// TIA Portal V20 program export: 1 tag tables, 0 data types, 3 data blocks, 33 code blocks (in call order from the OBs), 11 instance data blocks

VAR_GLOBAL   // PLC tag table "Default tag table"
   Doser1 AT %I0.0 : Bool;
   AlarmOpen1 AT %I0.1 : Bool;
   Doser2 AT %I0.2 : Bool;
   AlarmOpen2 AT %I0.3 : Bool;
   RunClose1 AT %I0.4 : Bool;
   RunOpen1 AT %I0.5 : Bool;
   RunClose2 AT %I0.6 : Bool;
   RunOpen2 AT %I0.7 : Bool;
   WaterCounterInPulse AT %I1.0 : Bool;
   WaterCounterOutPulse AT %I1.1 : Bool;
   AI0V AT %IW64 : Int;
   AI1V AT %IW66 : Int;
   AI0AV AT %IW128 : Int;
   AI1AV AT %IW130 : Int;
   AI2AV AT %IW132 : Int;
   AI3AV AT %IW134 : Int;
   AI4AV AT %IW80 : Int;
   PowerSupply AT %I1.2 : Bool;
   FlowAO AT %QW64 : Int;
   OutOpen1 AT %Q0.0 : Bool;
   OutClose1 AT %Q0.1 : Bool;
   OutOpen2 AT %Q0.2 : Bool;
   OutClose2 AT %Q0.3 : Bool;
   SirenOut AT %Q0.4 : Bool;
   System_Byte AT %MB1 : Byte;
   FirstScan AT %M1.0 : Bool;
   DiagStatusUpdate AT %M1.1 : Bool;
   AlwaysTRUE AT %M1.2 : Bool;
   AlwaysFALSE AT %M1.3 : Bool;
   Clock_Byte AT %MB0 : Byte;
   Clock_10Hz AT %M0.0 : Bool;
   Clock_5Hz AT %M0.1 : Bool;
   "Clock_2.5Hz" AT %M0.2 : Bool;
   Clock_2Hz AT %M0.3 : Bool;
   "Clock_1.25Hz" AT %M0.4 : Bool;
   Clock_1Hz AT %M0.5 : Bool;
   "Clock_0.625Hz" AT %M0.6 : Bool;
   "Clock_0.5Hz" AT %M0.7 : Bool;
   Damper1_AutoMode AT %I1.3 : Bool;
   Damper2_AutoMode AT %I1.4 : Bool;
   OsmosOut AT %Q0.5 : Bool;
   OsmosAO AT %QW66 : Int;
   DoserOut AT %Q0.6 : Bool;
   ChlorationOut AT %Q0.7 : Bool;
END_VAR

DATA_BLOCK "Config"   // DB20
{ S7_Optimized_Access := 'FALSE' }
VERSION : 0.1
// stored: AutoNumber false, DBAccessibleFromOPCUA true, IsOnlyStoredInLoadMemory false, IsWriteProtectedInAS false
   VAR
      DateTime : DTL := DTL#2024-10-30-11:20:02.078798;
      HMI_ResetWaterCounter : Bool := FALSE;
      HMI_ResetPositionDamper1 : Bool := FALSE;
      HMI_ResetPositionDamper2 : Bool := FALSE;
      HMI_StartAdjustDamper1 : Bool := FALSE;
      HMI_StartAdjustDamper2 : Bool := FALSE;
      HMI_StopAdjustDamper1 : Bool := FALSE;
      HMI_StopAdjustDamper2 : Bool := FALSE;
      HMI_WeightToZero : Bool := FALSE;
      WaterPulseDuble : Bool;
      DiOxydeDosing : DWord;
   END_VAR
BEGIN
END_DATA_BLOCK

DATA_BLOCK "MB"   // DB1
{ S7_Optimized_Access := 'FALSE' }
VERSION : 0.1
// stored: AutoNumber false, DBAccessibleFromOPCUA true, IsOnlyStoredInLoadMemory false, IsWriteProtectedInAS false
   VAR RETAIN
      Table : Struct
         Service : Bool := FALSE;
         CycleDay : Int := 0;
         CycleStatus : Word := 16#0001;
         RestTimeC1 : UInt := 10;
         RestTimeC2 : UInt := 20;
         RestTimeC3 : UInt := 27;
         RestTimeC4 : UInt := 45;
         RestTimeC5 : UInt := 9999;
         CycleStartDay : Array[0..4] of UInt;
         LevelRCV1Min : Real := 190.0;
         LevelRCV1Max : Real := 210.0;
         LevelRCV2Min : Real := 190.0;
         LevelRCV2Max : Real := 210.0;
         LevelRCV1BasicMin : Real := 200.0;
         LevelRCV1BasicMax : Real := 250.0;
         LevelRCV2BasicMin : Real := 200.0;
         LevelRCV2BasicMax : Real := 250.0;
         LevelRCVCycle : Array[0..4] of Struct
            Min : Real;
            Max : Real;
         END_STRUCT;
         WaterCounterInPulseValue : Real := 0.1;
         WaterCounterInDailyValue : Real := 0.0;
         WaterCounterInTotalValue : Real := 0.0;
         AIOffsetCH0 : Real := 0.0;
         AIValueMinCH0 : Real := 0.0;
         AIValueMaxCH0 : Real := 1.0;
         AITimeBaseCH0 : Time := T#0MS;
         AIOffsetCH1 : Real := 0.0;
         AIValueMinCH1 : Real := 0.0;
         AIValueMaxCH1 : Real := 1200.0;
         AITimeBaseCH1 : Time := T#5MS;
         AIOffsetCH2 : Real := 0.0;
         AIValueMinCH2 : Real := 0.0;
         AIValueMaxCH2 : Real := 1200.0;
         AITimeBaseCH2 : Time := T#5MS;
         AIOffsetCH3 : Real := 0.0;
         AIValueMinCH3 : Real := 0.0;
         AIValueMaxCH3 : Real := 16.0;
         AITimeBaseCH3 : Time := T#2MS;
         AIOffsetCH4 : Real := 0.0;
         AIValueMinCH4 : Real := 0.0;
         AIValueMaxCH4 : Real := 16.0;
         AITimeBaseCH4 : Time := T#2MS;
         AIOffsetCH5 : Real := 0.0;
         AIValueMinCH5 : Real := 0.0;
         AIValueMaxCH5 : Real := 0.0;
         AITimeBaseCH5 : Time := T#0MS;
         ChlorValue : Real := 0.8276128;
         RCV1LevelValue : Real := 0.07552084;
         RCV2LevelValue : Real := 199.1832;
         WaterInPressureValue : Real := 0.0;
         WaterOutPressureValue : Real := 4.414607;
         Reserved : Real := 0.0;
         LevelRCV1AlarmMin : Real := 100.0;
         LevelRCV1AlarmMax : Real := 400.0;
         LevelRCV2AlarmMin : Real := 100.0;
         LevelRCV2AlarmMax : Real := 400.0;
         Chlor_Setpoint : Real := 0.0;
         Chlor_PulseWeight : Real := 0.0;
         Chlor_ConcentAlarm : Real := 0.9;
         Chlor_BaseDose : Real := 25.0;   // Була задача в ручному
         Chlor_SetpointMin : Real := 1.0;
         Chlor_SetpointMax : Real := 1.1;
         Chlor_Corection : Real := 0.5;
         Doser1_PulseValue : Real := 10.0;
         Reserved_2 : Int := 0;
         Reserved_3 : Int := 0;
         Doser1_DailyValue : Real := 0.0;
         Doser1_TotalValue : Real := 0.0;
         Doser1_Cunsumption : Real := 0.0;
         Doser2_PulseValue : Real := 0.81;
         Reserved_4 : Int := 0;
         Reserved_5 : Int := 0;
         Doser2_DailyValue : Real := 0.0;
         Doser2_TotalValue : Real := 0.0;
         Doser2_Cunsumption : Real := 0.0;
         PumpDoserValue : Real := 0.0;
         CalibratedPumpDoserValueMA : Real := 4.0;
         PumpDoserCalibrationMA : Real := 0.0;
         PumpDoserProductivity : Real := 6300.0;
         DampersSyncMode : Word := 16#0000;
         UsePID : Bool := FALSE;
         Damper1_PID_SetpointDeadZone : Real := 5.0;
         Damper1_PID_KP : Real := 2.0;
         Damper1_PID_KI : Real := 0.3;
         Damper1_PID_KD : Real := 0.1;
         Damper1_PID_TI : Real := 600.0;
         Damper1_PositionDeadZone : Real := 1.0;
         Damper1_FullMovingTime : Real := 26.14;
         Damper1_Position : Real := 0.0;
         Damper1_PositionSetpoint : Real := 100.0;
         Damper1_PID_Setpoint : Real := 200.0;
         Damper2_PID_SetpointDeadZone : Real := 5.0;
         Damper2_PID_KP : Real := 2.0;
         Damper2_PID_KI : Real := 0.3;
         Damper2_PID_KD : Real := 0.1;
         Damper2_PID_TI : Real := 600.0;
         Damper2_PositionDeadZone : Real := 1.0;
         Damper2_FullMovingTime : Real := 28.0;
         Damper2_Position : Real := 0.0;
         Damper2_PositionSetpoint : Real := 0.0;
         Damper2_PID_Setpoint : Real := 200.0;
         HMI_CycleOn : Bool := TRUE;
         HMI_ChlorModeOn : Bool := FALSE;
         HMI_Chlor_ChooseTank : Bool := TRUE;   // 0 - РЧВ1 1 -РЧВ2
         HMI_ManualModeOn : Bool := FALSE;
         HMI_SoundOff : Bool := TRUE;
         HMI_ManualOpenDamper1 : Bool := FALSE;
         HMI_ManualOpenDamper2 : Bool := FALSE;
         HMI_ResetWaterCounter : Bool := FALSE;
         HMI_ResetPositionDamper1 : Bool := FALSE;
         HMI_ResetPositionDamper2 : Bool := FALSE;
         HMI_StartAdjustDamper1 : Bool := FALSE;
         HMI_StartAdjustDamper2 : Bool := FALSE;
         HMI_StopAdjustDamper1 : Bool := FALSE;
         HMI_StopAdjustDamper2 : Bool := FALSE;
         HMI_WeightToZero : Bool := FALSE;
         HMI_WeightAlarmReset : Bool := FALSE;
         Alarms_Open1 : Bool := FALSE;
         Alarms_Open2 : Bool := FALSE;
         Alarms_ChlorLargeConsumption : Bool := FALSE;
         Alarms_RCV1Max : Bool := FALSE;
         Alarms_RCV1Min : Bool := TRUE;
         Alarms_RCV2Max : Bool := FALSE;
         Alarms_RCV2Min : Bool := FALSE;
         Alarms_RCV1Error : Bool := FALSE;
         Alarms_RCV2Error : Bool := FALSE;
         Alarms_ChlorMax : Bool := FALSE;
         Alarms_NoFlow : Bool := FALSE;
         Alarms_WaterOutMax : Bool := FALSE;
         Alarms_WaterOutMin : Bool := FALSE;
         Alarms_NoPowerSupply : Bool := FALSE;
         Alarms_WaterInMax : Bool := FALSE;
         Alarms_WaterInMin : Bool := FALSE;
         WaterOutMaxValue : Real := 6.0;
         WaterOutMinValue : Real := 1.5;
         WaterOutAlarmTime : DInt := 10;
         GlobalAlarm : Bool := FALSE;
         SensorWeightVoltage1 : Real := 1.681112;
         WeightValueMin1 : Real := 356.0;
         WeightValueMax1 : Real := 361.0;
         WeightValueOffset1 : Real := 0.0;
         WeightValue1 : Real := 353.3342;
         WeightVoltageMin1 : Real := 1.691255;
         WeightVoltageMax1 : Real := 1.71028;
         DayChangeFlag : Bool := TRUE;
         Damper1_AdjustBusy : Bool := FALSE;
         Damper1_AdjustError : Bool := FALSE;
         Damper1_AdjustDone : Bool := FALSE;
         Damper2_AdjustBusy : Bool := FALSE;
         Damper2_AdjustError : Bool := FALSE;
         Damper2_AdjustDone : Bool := FALSE;
         "Damper1_Close/Open" : Bool := FALSE;
         "Damper2_Close/Open" : Bool := FALSE;
         "Damper1_Manual/Auto" : Bool := FALSE;
         "Damper2_Manual/Auto" : Bool := TRUE;
         SensorWeightVoltage2 : Real := -0.2375481;
         WeightValueMin2 : Real := 0.0;
         WeightValueMax2 : Real := 5.0;
         WeightValueOffset2 : Real := 0.0;
         WeightValue2 : Real := 0.0;
         WeightVoltageMin2 : Real := 0.155;
         WeightVoltageMax2 : Real := 0.177;
         WaterConsumption : Real := 0.0;
         LevelRCV1AlarmMinBasic : Real := 0.0;
         LevelRCV1AlarmMaxBasic : Real := 0.0;
         LevelRCV2AlarmMinBasic : Real := 0.0;
         LevelRCV2AlarmMaxBasic : Real := 0.0;
         LevelRCV1AlarmDeltaC1 : Real := 20.0;
         LevelRCV1AlarmDeltaC2 : Real := 20.0;
         LevelRCV1AlarmDeltaC3 : Real := 20.0;
         LevelRCV1AlarmDeltaC4 : Real := 20.0;
         LevelRCV1AlarmDeltaC5 : Real := 20.0;
         LevelRCV2AlarmDeltaC1 : Real := 20.0;
         LevelRCV2AlarmDeltaC2 : Real := 20.0;
         LevelRCV2AlarmDeltaC3 : Real := 20.0;
         LevelRCV2AlarmDeltaC4 : Real := 20.0;
         LevelRCV2AlarmDeltaC5 : Real := 20.0;
         WaterInPresMaxValue : Real := 8.0;
         WaterInPresMinValue : Real := 1.5;
         WaterInPresAlarmTime : DInt := 10;
         EndTag : Real := 0.0;
         WeightingEnable : Bool := TRUE;
         WeightingSetZero : Bool := FALSE;
         WeightValue1Liters : Real := 294.4452;
         WeightValue2Liters : Real := 0.0;
         WeightSensor1Error : Bool := FALSE;
         WeightSensor2Error : Bool := FALSE;
         Weighting_SaveManualValue : Bool := FALSE;
         Weighting_ManualValue1 : Real := 0.0;
         Weighting_ManualValue2 : Real := 0.0;
         WeightingDelay : DInt := 0;
         WeightingDeadZone : Real := 0.0;
         WeightingStat_CalendarMonth : Array[1..30] of UInt;
         WeightingStat_CalendarDay : Array[1..30] of UInt;
         WeightingStat_DayCycle : Array[1..30] of Int;
         WeightingStat_Counsumed1 : Array[1..30] of Real;
         WeightingStat_Load1 : Array[1..30] of Real;
         WeightingStat_Counsumed2 : Array[1..30] of Real;
         WeightingStat_Load2 : Array[1..30] of Real;
         ChlorReg_Update : Bool := FALSE;
         ChlorReg_DateTime : DTL := DTL#1970-01-01-00:00:00;
         HMI_ChlorReg_ValueRCV : Real := 0.0;
         HMI_ChlorReg_ValuePt : Real := 0.0;
         ChlorReg_ChlorValueRCV : Real := 0.0;
         ChlorReg_ChlorValuePt : Real := 0.0;
         ChlorReg_Age : Int := 0;
         Reserved_1 : Int := 0;
         ChlorReg_AgeF : Real := 0.0;
         WaterCounterIn_DailyCount : DInt := 0;
         WaterCounterIn_TotalCount : DInt := 0;
         Doser1_DailyPulses : DInt := 0;
         Doser1_TotalPulses : DInt := 0;
         Doser2_DailyPulses : DInt := 0;
         Doser2_TotalPulses : DInt := 0;
         WaterTemperature : Real := 18.22104;
         ChlorConsumptionTable : Array[0..3] of Struct
            Day : Int;
            MonitorTIme : Real;
            Consumption : Real;
         END_STRUCT;
         DoserNotWork : Bool := FALSE;
         Chlor_AutoMode : Bool := TRUE;
         Chlor_StartManual : Bool := FALSE;
         Chloration_ChooseCounter : Bool := FALSE;
         RecerculationFlow : Real := 0.0;
         FlowWithouRecerculation : Real := 17.51287;
         ChlorationParams : Struct
            SetpointMin : Real := 0.0;
            SetpointMax : Real := 0.0;
            BaseDose : Real := 0.0;
            ActualDose : Real := 0.0;
            DoseChangeMax : Real := 25.0;
            DosingMin : Real := 0.0;
            DosingMax : Real := 35.0;
            CorectionCoef : Real := 1.0;
         END_STRUCT;
         ChangeChlorMeasure : Bool := FALSE;
         MeasureChanged : Bool := FALSE;
         CriticalMeasureON : Bool := FALSE;
         MeasureNotEntered : Bool := FALSE;
         ChlorationCounter_SwitchOn : Bool := FALSE;
         ChlorMeasuredValue : Real := 0.0;
         ChlorMeasureTable : Array[0..3] of Struct
            CycleDay : Int;
            MeasureTime : Real;
            BlockTime : Real;
         END_STRUCT;
         TimeToMeasure : Real := 1.0;
         TimeToBlock : Real := 29.0;
         CriticalMeasure : Real := 1.5;
         Chlor_PulseWeight_1 : Real := 1.0;
         Chlor_ManualSetpoint_1 : Real := 0.0;
         MeasuredChlor : Real := 0.0;
         ClO2 : Struct
            AbsoluteDosing : Real := 0.0;
            ProportionalDosingEmbedded : Real := 0.0;
            ProportionalDosingExternal : Real := 0.0;
            ChooseDosing : Word := 16#1204;
            DosersActive : Word := 16#0006;
            WorkMode : Word := 16#0001;
            Doser1Productivity : Real := 0.0;
            Doser2Productivity : Real := 0.0;
            Pressure : Real := 0.0;
            SystemProductivity : Real := 0.0;
            Alarms : Word := 16#0000;
         END_STRUCT;
         WaterCounterOut_DailyCount : DInt := 3;
         WaterCounterOut_TotalCount : DInt := 3;
         WaterCounterOut_DailyValue : Real := 0.3;
         WaterCounterOut_TotalValue : Real := 0.3;
         WaterCounterOut_PulseValue : Real := 0.1;
         WaterCounterOut_Consumption : Real := 16#7F80_0000;
         ChlorationCounter_SwitchDay : Int := 5;
         END : Array[0..10] of Word;
      END_STRUCT;
   END_VAR
BEGIN
   Table.CycleStartDay[0] := 0;
   Table.CycleStartDay[1] := 10;
   Table.CycleStartDay[2] := 20;
   Table.CycleStartDay[3] := 27;
   Table.CycleStartDay[4] := 45;
   Table.LevelRCVCycle[0].Min := 190.0;
   Table.LevelRCVCycle[1..3].Min := 270.0;
   Table.LevelRCVCycle[4].Min := 190.0;
   Table.LevelRCVCycle[0].Max := 210.0;
   Table.LevelRCVCycle[1..3].Max := 310.0;
   Table.LevelRCVCycle[4].Max := 210.0;
   Table.WeightingStat_CalendarMonth[1] := 7;
   Table.WeightingStat_CalendarMonth[2..30] := 0;
   Table.WeightingStat_CalendarDay[1] := 7;
   Table.WeightingStat_CalendarDay[2..30] := 0;
   Table.WeightingStat_DayCycle[1..30] := 0;
   Table.WeightingStat_Counsumed1[1] := 0.0133667;
   Table.WeightingStat_Counsumed1[2..30] := 0.0;
   Table.WeightingStat_Load1[1] := 353.3476;
   Table.WeightingStat_Load1[2..30] := 0.0;
   Table.WeightingStat_Counsumed2[1..30] := 0.0;
   Table.WeightingStat_Load2[1..30] := 0.0;
   Table.ChlorConsumptionTable[0].Day := 0;
   Table.ChlorConsumptionTable[1].Day := 6;
   Table.ChlorConsumptionTable[2].Day := 18;
   Table.ChlorConsumptionTable[3].Day := 30;
   Table.ChlorConsumptionTable[0..3].MonitorTIme := 1.0;
   Table.ChlorConsumptionTable[0..3].Consumption := 3.0;
   Table.ChlorMeasureTable[0..3].CycleDay := 0;
   Table.ChlorMeasureTable[0..3].MeasureTime := 1.0;
   Table.ChlorMeasureTable[0..3].BlockTime := 29.0;
   Table.END[0..10] := 16#0000;
END_DATA_BLOCK

DATA_BLOCK "MB_Config"   // DB14
{ S7_Optimized_Access := 'TRUE' }
VERSION : 0.1
// stored: AutoNumber true, DBAccessibleFromOPCUA true, IsOnlyStoredInLoadMemory false, IsRetainMemResEnabled false, IsWriteProtectedInAS false, MemoryReserve 100
   VAR
      CONNECT : TCON_IP_v4;
      NDR : Bool := FALSE;
      DR : Bool := FALSE;
      ERROR : Bool := FALSE;
      STATUS : Word := 16#0000;
      BUFFER : Array[0..500] of Word;
   END_VAR
BEGIN
   CONNECT.InterfaceId := 64;
   CONNECT.ID := 16#0001;
   CONNECT.ConnectionType := 16#0B;
   CONNECT.ActiveEstablished := FALSE;
   CONNECT.RemoteAddress.ADDR[1..4] := 16#00;
   CONNECT.RemotePort := 0;
   CONNECT.LocalPort := 502;
   BUFFER[0..500] := 16#0000;
END_DATA_BLOCK

ORGANIZATION_BLOCK "Main"   // OB1, SCL, ProgramCycle
TITLE = "Main Program Sweep (Cycle)"
{ S7_Optimized_Access := 'TRUE' }
VERSION : 0.1
// stored: AutoNumber true, IsIECCheckEnabled false, SetENOAutomatically false
   VAR_INPUT
      Initial_Call : Bool;   // Initial call of this OB
      Remanence : Bool;   // =True, if remanent data are available
   END_VAR
BEGIN
   "SystemClock"();
   "Inputs_DB"();
   "WaterCounter_DB"();
   "HMI_DB"();
   "Alarms_DB"();
   "WorkModeCycle_DB"();
   "Dampers_DB"();
   "Weighting_DB"();
   "MBServer_DB"();
   "ModbusClO2_DB"();
   "ChlorMode_DB"();

   "MB".Table.Chlor_Setpoint := "MB".Table.ChlorationParams.ActualDose;
   "MB".Table.Chlor_PulseWeight := "MB".Table.MeasuredChlor;
END_ORGANIZATION_BLOCK

FUNCTION_BLOCK "Inputs"   // FB4, SCL
{ S7_Optimized_Access := 'TRUE' }
VERSION : 0.1
// stored: AutoNumber true, IsIECCheckEnabled false, IsRetainMemResEnabled false, MemoryReserve 100, SetENOAutomatically false, UDAEnableTagReadback false
   VAR
      AIHandlers { S7_SetPoint := 'True'} : Array[0..5] of "AIHandler";
      WeightHandlers { S7_SetPoint := 'True'} : Array[0..1] of "WeightHandler";
      ErrorRCV1 { S7_SetPoint := 'True'} : Bool;
      ErrorRCV2 { S7_SetPoint := 'True'} : Bool;
   END_VAR
BEGIN
   #AIHandlers[0](
                  Value := "AI0AV",
                  ValueMin := 0,
                  ValueMax := 27648,
                  ValueOffset := "MB".Table.AIOffsetCH0,
                  OutputMin := "MB".Table.AIValueMinCH0,
                  OutputMax := "MB".Table.AIValueMaxCH0,
                  TimeBase := "MB".Table.AITimeBaseCH0,
                  Output => "MB".Table.WaterInPressureValue);
   #AIHandlers[1](
                  Value := "AI1AV",
                  ValueMin := 0,
                  ValueMax := 27648,
                  ValueOffset := "MB".Table.AIOffsetCH1,
                  OutputMin := "MB".Table.AIValueMinCH1,
                  OutputMax := "MB".Table.AIValueMaxCH1,
                  TimeBase := "MB".Table.AITimeBaseCH1,
                  Output => "MB".Table.RCV1LevelValue);
   #AIHandlers[2](
                  Value := "AI2AV",
                  ValueMin := 0,
                  ValueMax := 27648,
                  ValueOffset := "MB".Table.AIOffsetCH2,
                  OutputMin := "MB".Table.AIValueMinCH2,
                  OutputMax := "MB".Table.AIValueMaxCH2,
                  TimeBase := "MB".Table.AITimeBaseCH2,
                  Output => "MB".Table.RCV2LevelValue);
   #AIHandlers[3](
                  Value := "AI3AV",
                  ValueMin := 0,
                  ValueMax := 27648,
                  ValueOffset := "MB".Table.AIOffsetCH3,
                  OutputMin := "MB".Table.AIValueMinCH3,
                  OutputMax := "MB".Table.AIValueMaxCH3,
                  TimeBase := "MB".Table.AITimeBaseCH3,
                  Output => "MB".Table.WaterOutPressureValue);
   // #AIHandlers[4](
   //                Value := "AI4AV",
   //                ValueMin := 5320,
   //                ValueMax := 27648,
   //                ValueOffset := "MB".Table.AIOffsetCH4,
   //                OutputMin := "MB".Table.AIValueMinCH4,
   //                OutputMax := "MB".Table.AIValueMaxCH4,
   //                TimeBase := "MB".Table.AITimeBaseCH4,
   //                Output => );

   #ErrorRCV1 := #AIHandlers[1].Error;
   #ErrorRCV2 := #AIHandlers[2].Error;


   CASE "MB".Table.DampersSyncMode OF
       1:
           "MB".Table.RCV1LevelValue := "MB".Table.RCV1LevelValue;
           "MB".Table.RCV2LevelValue := "MB".Table.RCV1LevelValue;
           #ErrorRCV2 := #ErrorRCV1;
       2:
           "MB".Table.RCV1LevelValue := "MB".Table.RCV2LevelValue;
           "MB".Table.RCV2LevelValue := "MB".Table.RCV2LevelValue;
           #ErrorRCV1 := #ErrorRCV2;
   END_CASE;
END_FUNCTION_BLOCK

FUNCTION_BLOCK "AIHandler"   // FB3, SCL
{ S7_Optimized_Access := 'TRUE' }
VERSION : 0.1
// stored: AutoNumber true, IsIECCheckEnabled false, IsRetainMemResEnabled false, MemoryReserve 100, SetENOAutomatically false, UDAEnableTagReadback false
   VAR_INPUT
      Value : Real;
      ValueMin : Real;
      ValueMax : Real;
      ValueOffset : Real;
      OutputMin : Real;
      OutputMax : Real;
      TimeBase : Time := T#1s;
   END_VAR
   VAR_OUTPUT
      Output : Real;
      Error : Bool;
   END_VAR
   VAR
      ConvertedValue : Real;
      TON1 { S7_SetPoint := 'True'} : TON_TIME;
      DelayTON { S7_SetPoint := 'True'} : TON_TIME;
      FilterArray : Array[0..199] of Real;
      FilterTime : Time;
      i : Int;
      sum : Real;
      FilteredValue : Real;
      one : Bool;
   END_VAR
   VAR CONSTANT
      TimeDelay : Time := T#120s;
   END_VAR
BEGIN

   #FilterTime := #TimeBase * 1000 /50;

   #DelayTON(IN := TRUE,
             PT := #FilterTime);


   IF #DelayTON.Q = TRUE THEN
           RESET_TIMER(#DelayTON);
           #sum := #sum + #Value;
           #i := #i + 1;
           IF (#i >= 50) THEN
               #i := 0;
               #FilteredValue := #sum / 50.0;
               #ConvertedValue := (#FilteredValue - #ValueMin) / (#ValueMax - #ValueMin) * (#OutputMax - #OutputMin) + #OutputMin;
               #sum := 0;
               IF (#ConvertedValue < 0) THEN
                   #Output := 0;
               ELSE
                   #Output := #ConvertedValue + #ValueOffset;
               END_IF;
           END_IF;
   END_IF;

   #TON1(IN := #Value > 30000,
         PT := #TimeDelay,
         Q => #Error);
END_FUNCTION_BLOCK

FUNCTION_BLOCK "WaterCounter"   // FB1, SCL
{ S7_Optimized_Access := 'TRUE' }
VERSION : 0.1
// stored: AutoNumber true, IsIECCheckEnabled false, IsRetainMemResEnabled false, MemoryReserve 100, SetENOAutomatically false, UDAEnableTagReadback false
   VAR
      WaterCounter_InWater : "FlowCounter";
      WaterCounter_OutWater : "FlowCounter";
      DelayTON { S7_SetPoint := 'True'} : TON_TIME;
      ChlorCounter_1 { S7_SetPoint := 'True'} : "FlowCounter";
      ChlorCounter_2 { S7_SetPoint := 'True'} : "FlowCounter";
   END_VAR
BEGIN
   #WaterCounter_InWater(Pulse:="WaterCounterInPulse",
                         DailyCount:="MB".Table.WaterCounterIn_DailyCount,
                         TotalCount:="MB".Table.WaterCounterIn_TotalCount,
                         PulseWeight:="MB".Table.WaterCounterInPulseValue,
                         Consumption:="MB".Table.WaterConsumption,
                         DailyValue:="MB".Table.WaterCounterInDailyValue,
                         TotalValue:="MB".Table.WaterCounterInTotalValue);

   #WaterCounter_OutWater(Pulse := "WaterCounterOutPulse",
                          DailyCount := "MB".Table.WaterCounterOut_DailyCount,
                          TotalCount := "MB".Table.WaterCounterOut_TotalCount,
                          PulseWeight := "MB".Table.WaterCounterOut_PulseValue,
                          Consumption := "MB".Table.WaterCounterOut_Consumption,
                          DailyValue := "MB".Table.WaterCounterOut_DailyValue,
                          TotalValue := "MB".Table.WaterCounterOut_TotalValue);

   IF #WaterCounter_OutWater.R_TRIG_Instance.Q THEN
       "Config".WaterPulseDuble := TRUE;
   END_IF;



   IF NOT "MB".Table.Chloration_ChooseCounter THEN
       "ChlorationOut" := "WaterCounterOutPulse";
   ELSE
       "ChlorationOut" := "WaterCounterInPulse";
   END_IF;

   IF "MB".Table.WaterCounterOut_Consumption < 0 THEN
       "FlowAO" := 5520;
   ELSIF "MB".Table.WaterCounterOut_Consumption > 80.0 THEN
       "FlowAO" := 27648;
   ELSE
       "FlowAO" := REAL_TO_INT(("MB".Table.WaterCounterOut_Consumption) / (80) * (27648 - 5520) + 5520);
   END_IF;

   // IF "MB".Table.WaterConsumption < 0 THEN
   //     "OsmosAO" := 5520;
   // ELSIF "MB".Table.WaterConsumption > 80.0 THEN
   //     "OsmosAO" := 27648;
   // ELSE
   //     "OsmosAO" := REAL_TO_INT(("MB".Table.WaterConsumption - "MB".Table.RecerculationFlow) / (80) * (27648 - 5520) + 5520);
   // END_IF;
   // "MB".Table.FlowWithouRecerculation := "MB".Table.WaterConsumption - "MB".Table.RecerculationFlow;
   // IF "MB".Table.FlowWithouRecerculation < 0 THEN
   //     "MB".Table.FlowWithouRecerculation := 0;
   // END_IF;


   #ChlorCounter_1(Pulse:="Doser1",
                   DailyCount:="MB".Table.Doser1_DailyPulses,
                   TotalCount:="MB".Table.Doser1_TotalPulses,
                  PulseWeight:="MB".Table.Doser1_PulseValue,
                  Consumption := "MB".Table.Doser1_Cunsumption,
                  DailyValue:="MB".Table.Doser1_DailyValue,
                  TotalValue:="MB".Table.Doser1_TotalValue);

   #ChlorCounter_2(Pulse := "Doser2",
                   DailyCount := "MB".Table.Doser2_DailyPulses,
                   TotalCount := "MB".Table.Doser2_TotalPulses,
                  PulseWeight := "MB".Table.Doser2_PulseValue,
                  Consumption := "MB".Table.Doser2_Cunsumption,
                  DailyValue := "MB".Table.Doser2_DailyValue,
                  TotalValue := "MB".Table.Doser2_TotalValue);
END_FUNCTION_BLOCK

FUNCTION_BLOCK "FlowCounter"   // FB27, SCL
{ S7_Optimized_Access := 'TRUE' }
VERSION : 0.1
// stored: AutoNumber true, IsIECCheckEnabled false, IsRetainMemResEnabled false, MemoryReserve 100, SetENOAutomatically false, UDAEnableTagReadback false
   VAR_IN_OUT
      Pulse : Bool;
      DailyCount : DInt;
      TotalCount : DInt;
      PulseWeight : Real;
      Consumption : Real;
      DailyValue : Real;
      TotalValue : Real;
   END_VAR
   VAR
      R_TRIG_Instance { S7_SetPoint := 'True'} : R_TRIG;
      HourTimer { S7_SetPoint := 'True'} : TON_TIME;
      PrevValue { S7_SetPoint := 'True'} : Real;
      TimeNow : DTL;
      TimeLast : DTL;
      Ret : Int;
      TimeDif : Time;
      FilterArr : Array[0..3] of Real;
      i : Int;
      NoFlowTON { S7_SetPoint := 'True'} : TON_TIME;
   END_VAR
   VAR_TEMP
      j : Int;
      sum : Real;
   END_VAR
BEGIN
   #R_TRIG_Instance(CLK := #Pulse,
                    Q => #R_TRIG_Instance.Q);

   #HourTimer.TON(IN := TRUE,
   PT := T#3600s);

   #NoFlowTON(IN := TRUE,
              PT := T#300s);

   IF #R_TRIG_Instance.Q THEN
       RESET_TIMER(#NoFlowTON);
       #R_TRIG_Instance.CLK := FALSE;
       IF (#i > 3) THEN
           #i := 0;
       END_IF;

       #DailyCount += 1;
       #TotalCount += 1;
       #Ret := RD_SYS_T(#TimeNow);
       #TimeDif := #TimeNow - #TimeLast;
       #FilterArr[#i] := 3600 * 1000 / DINT_TO_REAL(#TimeDif) * #PulseWeight;
       FOR #j := 0 TO 3 DO
           #sum += #FilterArr[#j];
       END_FOR;

       #Consumption := #sum / 4;
       #TimeLast := #TimeNow;
       #i += 1;
       #sum := 0;

   END_IF;

   #DailyValue := UDINT_TO_REAL(#DailyCount) * #PulseWeight;
   #TotalValue := UDINT_TO_REAL(#TotalCount) * #PulseWeight;

   IF #NoFlowTON.Q THEN
       #Consumption := 0;
   END_IF;

   IF "Config".HMI_ResetWaterCounter THEN
       #DailyCount := 0;
       #TotalCount := 0;
   END_IF;
END_FUNCTION_BLOCK

FUNCTION_BLOCK "HMI"   // FB16, SCL
{ S7_Optimized_Access := 'TRUE' }
VERSION : 0.1
// stored: AutoNumber true, IsIECCheckEnabled false, IsRetainMemResEnabled false, MemoryReserve 100, SetENOAutomatically false, UDAEnableTagReadback false
   VAR
      UpdateTimer { S7_SetPoint := 'True'} : TON_TIME;
   END_VAR
   VAR_TEMP
      Ret : Int;
   END_VAR
BEGIN
   "Config".HMI_ResetWaterCounter := "MB".Table.HMI_ResetWaterCounter;
   IF "MB".Table.HMI_ResetWaterCounter THEN
       "MB".Table.HMI_ResetWaterCounter := 0;
   END_IF;

   "Config".HMI_ResetPositionDamper1 := "MB".Table.HMI_ResetPositionDamper1;
   IF "MB".Table.HMI_ResetPositionDamper1 THEN
       "MB".Table.HMI_ResetPositionDamper1 := 0;
   END_IF;

   "Config".HMI_ResetPositionDamper2 := "MB".Table.HMI_ResetPositionDamper2;
   IF "MB".Table.HMI_ResetPositionDamper2 THEN
       "MB".Table.HMI_ResetPositionDamper2 := 0;
   END_IF;

   "Config".HMI_StartAdjustDamper1 := "MB".Table.HMI_StartAdjustDamper1;
   IF "MB".Table.HMI_StartAdjustDamper1 THEN
       "MB".Table.HMI_StartAdjustDamper1 := 0;
   END_IF;

   "Config".HMI_StartAdjustDamper2 := "MB".Table.HMI_StartAdjustDamper2;
   IF "MB".Table.HMI_StartAdjustDamper2 THEN
       "MB".Table.HMI_StartAdjustDamper2 := 0;
   END_IF;

   "Config".HMI_StopAdjustDamper1 := "MB".Table.HMI_StopAdjustDamper1;
   IF "MB".Table.HMI_StopAdjustDamper1 THEN
       "MB".Table.HMI_StopAdjustDamper1 := 0;
   END_IF;

   "Config".HMI_StopAdjustDamper2 := "MB".Table.HMI_StopAdjustDamper2;
   IF "MB".Table.HMI_StopAdjustDamper2 THEN
       "MB".Table.HMI_StopAdjustDamper2 := 0;
   END_IF;

   "Config".HMI_WeightToZero := "MB".Table.HMI_WeightToZero;
   IF "MB".Table.HMI_WeightToZero THEN
       "MB".Table.HMI_WeightToZero := 0;
   END_IF;

   IF "MB".Table.ChlorReg_Update THEN
       "MB".Table.ChlorReg_ChlorValueRCV := "MB".Table.HMI_ChlorReg_ValueRCV;
       "MB".Table.ChlorReg_ChlorValuePt := "MB".Table.HMI_ChlorReg_ValuePt;
       "MB".Table.ChlorReg_Age := "MB".Table.CycleDay;
       "MB".Table.ChlorReg_AgeF := INT_TO_REAL("MB".Table.CycleDay);
       #Ret:= RD_SYS_T("MB".Table.ChlorReg_DateTime);
       #UpdateTimer(IN:=TRUE,
                    PT:=T#100ms);
       IF #UpdateTimer.Q THEN
           "MB".Table.ChlorReg_Update := FALSE;
           RESET_TIMER(#UpdateTimer);
       END_IF;


   END_IF;
END_FUNCTION_BLOCK

FUNCTION_BLOCK "Alarms"   // FB17, SCL
{ S7_Optimized_Access := 'TRUE' }
VERSION : 0.1
// stored: AutoNumber true, IsIECCheckEnabled false, IsRetainMemResEnabled false, MemoryReserve 100, SetENOAutomatically false, UDAEnableTagReadback false
   VAR
      WaterOutMaxTON { S7_SetPoint := 'True'} : TON_TIME;
      WaterOutMinTON { S7_SetPoint := 'True'} : TON_TIME;
      WaterInMaxTON { S7_SetPoint := 'True'} : TON_TIME;
      WaterInMinTON { S7_SetPoint := 'True'} : TON_TIME;
      "step" { S7_SetPoint := 'True'} : Int;
      ChlorAlarm { S7_SetPoint := 'True'} : "ChlorConsumptionAlarm";
   END_VAR
BEGIN
   #step := 0;
   "MB".Table.Alarms_Open1:="AlarmOpen1";
   "MB".Table.Alarms_Open2:="AlarmOpen2";

   "MB".Table.Alarms_RCV1Max:="MB".Table.RCV1LevelValue>="MB".Table.LevelRCV1AlarmMax;
   "MB".Table.Alarms_RCV1Min:="MB".Table.RCV1LevelValue<="MB".Table.LevelRCV1AlarmMin;
   "MB".Table.Alarms_RCV2Max:="MB".Table.RCV2LevelValue>="MB".Table.LevelRCV2AlarmMax;
   "MB".Table.Alarms_RCV2Min:="MB".Table.RCV2LevelValue<="MB".Table.LevelRCV2AlarmMin;

   "MB".Table.Alarms_RCV1Error:="Inputs_DB".ErrorRCV1;
   "MB".Table.Alarms_RCV2Error:="Inputs_DB".ErrorRCV2;

   "MB".Table.Alarms_ChlorMax:="MB".Table.ChlorValue>="MB".Table.Chlor_ConcentAlarm;

   //"MB".Table.Alarms_NoFlow:= NOT("FlowSensor");

   "MB".Table.Alarms_NoPowerSupply:= NOT ("PowerSupply");

   #WaterOutMaxTON(IN := "MB".Table.WaterOutPressureValue >= "MB".Table.WaterOutMaxValue,
                   PT := "MB".Table.WaterOutAlarmTime * 1000);
   "MB".Table.Alarms_WaterOutMax := #WaterOutMaxTON.Q;

   #WaterOutMinTON(IN:="MB".Table.WaterOutPressureValue<="MB".Table.WaterOutMinValue,
                   PT:="MB".Table.WaterOutAlarmTime*1000);
   "MB".Table.Alarms_WaterOutMin := #WaterOutMinTON.Q;

   #WaterInMaxTON(IN:="MB".Table.WaterInPressureValue >= "MB".Table.WaterInPresMaxValue,
                  PT:="MB".Table.WaterInPresAlarmTime*1000);
   "MB".Table.Alarms_WaterInMax := #WaterInMaxTON.Q;

   #WaterInMinTON(IN:="MB".Table.WaterInPressureValue <= "MB".Table.WaterInPresMinValue,
                  PT:="MB".Table.WaterInPresAlarmTime*1000);

   #ChlorAlarm(HighAlarm=>"MB"  .Table.Alarms_ChlorLargeConsumption);


   "MB".Table.Alarms_WaterInMin := #WaterOutMinTON.Q;

   "SirenOut" := %DB1. > 0 AND NOT "MB".Table.HMI_SoundOff;
END_FUNCTION_BLOCK

FUNCTION_BLOCK "ChlorConsumptionAlarm"   // FB6, SCL
{ S7_Optimized_Access := 'TRUE' }
VERSION : 0.1
// stored: AutoNumber true, IsIECCheckEnabled false, IsRetainMemResEnabled false, MemoryReserve 100, SetENOAutomatically false, UDAEnableTagReadback false
   VAR_OUTPUT
      HighAlarm : Bool;
   END_VAR
   VAR
      "step" : Int;
      maxConsamption : Real;
      monitorTime : Real;
      weightNow : Real;
      weightLast : Real;
      TON { S7_SetPoint := 'True'} : TON_TIME;
      weightDelta { S7_SetPoint := 'True'} : Real;
   END_VAR
BEGIN
   #maxConsamption := "MB".Table.ChlorConsumptionTable[0].Consumption;
   #monitorTime := "MB".Table.ChlorConsumptionTable[0].MonitorTIme;

   IF "MB".Table.CycleDay >= "MB".Table.ChlorConsumptionTable[3].Day THEN
       #maxConsamption := "MB".Table.ChlorConsumptionTable[3].Consumption;
       #monitorTime    := "MB".Table.ChlorConsumptionTable[3].MonitorTIme;
   ELSIF "MB".Table.CycleDay >= "MB".Table.ChlorConsumptionTable[2].Day THEN
       #maxConsamption := "MB".Table.ChlorConsumptionTable[2].Consumption;
       #monitorTime    := "MB".Table.ChlorConsumptionTable[2].MonitorTIme;
   ELSIF "MB".Table.CycleDay >= "MB".Table.ChlorConsumptionTable[1].Day THEN
       #maxConsamption := "MB".Table.ChlorConsumptionTable[1].Consumption;
       #monitorTime    := "MB".Table.ChlorConsumptionTable[1].MonitorTIme;
   ELSIF "MB".Table.CycleDay >= "MB".Table.ChlorConsumptionTable[0].Day THEN
       #maxConsamption := "MB".Table.ChlorConsumptionTable[0].Consumption;
       #monitorTime    := "MB".Table.ChlorConsumptionTable[0].MonitorTIme;
   END_IF;

   #TON(IN:=TRUE,
        PT:=REAL_TO_DINT(#monitorTime*3600*1000));

   IF #TON.Q THEN
       #weightLast := #weightNow;
       RESET_TIMER(#TON);
   END_IF;
   #weightNow := "MB".Table.WeightValue1Liters;
   #weightDelta := #weightLast - #weightNow;


   IF "MB".Table.HMI_WeightAlarmReset THEN
       #weightDelta := 0;
       #weightNow := "MB".Table.WeightValue1Liters;
       #weightLast := #weightNow;
       #HighAlarm := false;
       RESET_TIMER(#TON);
       "MB".Table.HMI_WeightAlarmReset := FALSE;
   END_IF;

   IF #weightDelta > #maxConsamption THEN
       #HighAlarm := TRUE;
   END_IF;
END_FUNCTION_BLOCK

FUNCTION_BLOCK "WorkModeCycle"   // FB2, SCL
{ S7_Optimized_Access := 'TRUE' }
VERSION : 0.1
// stored: AutoNumber true, IsIECCheckEnabled false, IsRetainMemResEnabled false, MemoryReserve 100, SetENOAutomatically false, UDAEnableTagReadback false
   VAR
      "step" : Int;
      tod : Time_Of_Day;
      "return" : Int;
      dtl : DTL;
      "time" : Time;
      fracDay : Real;
   END_VAR
BEGIN
   #step := 0;

   "MB".Table.LevelRCV1Min:="MB".Table.LevelRCV1BasicMin;
   "MB".Table.LevelRCV1Max:="MB".Table.LevelRCV1BasicMax;
   "MB".Table.LevelRCV2Min:="MB".Table.LevelRCV2BasicMin;
   "MB".Table.LevelRCV2Max:="MB".Table.LevelRCV2BasicMax;

   "MB".Table.CycleStatus := 0;

   "MB".Table.RestTimeC1 := 0;
   "MB".Table.RestTimeC2 := 0;
   "MB".Table.RestTimeC3 := 0;
   "MB".Table.RestTimeC4 := 0;
   "MB".Table.RestTimeC5 := 0;

   #return := RD_LOC_T(#dtl);
   #tod := DTL_TO_TOD(#dtl);
   #time := TOD_TO_TIME(#tod);

   #fracDay := DINT_TO_REAL(#time) / 86400000.0;

   IF "MB".Table.HMI_CycleOn THEN
       IF "MB".Table.CycleDay >= "MB".Table.CycleStartDay[4] THEN
           #step := 4;
           "MB".Table.CycleStatus.%X4 := 1;
       ELSIF "MB".Table.CycleDay >= "MB".Table.CycleStartDay[3] THEN
           #step := 3;
           "MB".Table.CycleStatus.%X3 := 1;
       ELSIF "MB".Table.CycleDay >= "MB".Table.CycleStartDay[2] THEN
           #step := 2;
           "MB".Table.CycleStatus.%X2 := 1;
       ELSIF "MB".Table.CycleDay>="MB".Table.CycleStartDay[1] THEN
           #step := 1;
           "MB".Table.CycleStatus.%X1 := 1;
       ELSE
           #step := 0;
           "MB".Table.CycleStatus.%X0 := 1;
       END_IF;




       "MB".Table.LevelRCV1Min := "MB".Table.LevelRCVCycle[#step].Min;
       "MB".Table.LevelRCV2Min := "MB".Table.LevelRCVCycle[#step].Min;
       "MB".Table.LevelRCV1Max := "MB".Table.LevelRCVCycle[#step].Max;
       "MB".Table.LevelRCV2Max := "MB".Table.LevelRCVCycle[#step].Max;

       IF #step <> 4 THEN
           IF "MB".Table.CycleStartDay[#step + 1] - "MB".Table.CycleDay = 1 THEN
               "MB".Table.LevelRCV1Min := #fracDay * ("MB".Table.LevelRCVCycle[#step + 1].Min - "MB".Table.LevelRCVCycle[#step].Min) + "MB".Table.LevelRCVCycle[#step].Min;
               "MB".Table.LevelRCV1Max := #fracDay * ("MB".Table.LevelRCVCycle[#step + 1].Max - "MB".Table.LevelRCVCycle[#step].Max) + "MB".Table.LevelRCVCycle[#step].Max;
               "MB".Table.LevelRCV2Min := #fracDay * ("MB".Table.LevelRCVCycle[#step + 1].Min - "MB".Table.LevelRCVCycle[#step].Min) + "MB".Table.LevelRCVCycle[#step].Min;
               "MB".Table.LevelRCV2Max := #fracDay * ("MB".Table.LevelRCVCycle[#step + 1].Max - "MB".Table.LevelRCVCycle[#step].Max) + "MB".Table.LevelRCVCycle[#step].Max;
           END_IF;
       END_IF;



       "MB".Table.RestTimeC1:= MAX(IN1 :="MB".Table.CycleStartDay[1]-"MB".Table.CycleDay, IN2 := 0);
       "MB".Table.RestTimeC2:= MAX(IN1 :="MB".Table.CycleStartDay[2]-"MB".Table.CycleDay, IN2 := 0);
       "MB".Table.RestTimeC3:= MAX(IN1 :="MB".Table.CycleStartDay[3]-"MB".Table.CycleDay, IN2 := 0);
       "MB".Table.RestTimeC4:= MAX(IN1 :="MB".Table.CycleStartDay[4]-"MB".Table.CycleDay, IN2 := 0);
       "MB".Table.RestTimeC5 := 9999;
   END_IF;
END_FUNCTION_BLOCK

FUNCTION_BLOCK "Dampers"   // FB15, SCL
{ S7_Optimized_Access := 'TRUE' }
VERSION : 0.1
// stored: AutoNumber true, IsIECCheckEnabled false, IsRetainMemResEnabled false, MemoryReserve 100, SetENOAutomatically false, UDAEnableTagReadback false
   VAR
      DamperController1 { S7_SetPoint := 'True'} : "DamperController";
      DamperController2 { S7_SetPoint := 'True'} : "DamperController";
      DamperController3 { S7_SetPoint := 'True'} : "DamperController";
   END_VAR
BEGIN
   IF "Inputs_DB".ErrorRCV1 THEN
       #DamperController1.ManualMode := TRUE;
       #DamperController1.ManaulOpen := FALSE;
       #DamperController1.ManualClose := TRUE;
   ELSE
       #DamperController1.ManualMode := "MB".Table.HMI_ManualModeOn;
       #DamperController1.ManaulOpen := "MB".Table.HMI_ManualOpenDamper1;
       #DamperController1.ManualClose := NOT "MB".Table.HMI_ManualOpenDamper1;
   END_IF;

   #DamperController1(TankLevel:="MB".Table.RCV1LevelValue,
                      TankLevelSetpoint:=("MB".Table.LevelRCV1Min + ("MB".Table.LevelRCV1Max-"MB".Table.LevelRCV1Min)/2),
                      TankLevelMin:="MB".Table.LevelRCV1Min,
                      TankLevelMax:="MB".Table.LevelRCV1Max,
                      UsePID:="MB".Table.UsePID,
                      PID_DeadZone:="MB".Table.Damper1_PID_SetpointDeadZone,
                      PID_KP:="MB".Table.Damper1_PID_KP,
                      PID_KI:="MB".Table.Damper1_PID_KI,
                      PID_KD:="MB".Table.Damper1_PID_KD,
                      PID_TI:="MB".Table.Damper1_PID_TI,
                      LimitSwitch0:="RunClose1",
                      LimitSwitch100:="RunOpen1",
                      PouseMove:=5,
                      PositionDeadzone:="MB".Table.Damper1_PositionDeadZone,
                      StartAjustment:="Config".HMI_StartAdjustDamper1,
                      CancelAjustment:="Config".HMI_StopAdjustDamper1,
                      ResetPosition:="Config".HMI_ResetPositionDamper1,
                      Open=>"OutOpen1",
                      Close=>"OutClose1",
                      FullMovingTime:="MB".Table.Damper1_FullMovingTime,
                      SwitchAutoMode := "Damper1_AutoMode");

   "MB".Table."Damper1_Manual/Auto" := "Damper1_AutoMode";

   "MB".Table.Damper1_Position := #DamperController1.CurrentPosition;
   "MB".Table.Damper1_PositionSetpoint := #DamperController1.PositionSetPoint;
   "MB".Table.Damper1_PID_Setpoint := #DamperController1.TankLevelSetpoint;
   "MB".Table.Damper1_AdjustBusy := #DamperController1.AdjustBusy;
   "MB".Table.Damper1_AdjustError := #DamperController1.AdjustError;
   "MB".Table.Damper1_AdjustDone := WORD_TO_BOOL(#DamperController1.AdjustmentDone);

   IF "MB".Table.Damper1_Position > 0 THEN
       "MB".Table."Damper1_Close/Open" := TRUE;
   ELSE
       "MB".Table."Damper1_Close/Open" := FALSE;
   END_IF;

   IF "Inputs_DB".ErrorRCV2 THEN
       #DamperController2.ManualMode := TRUE;
       #DamperController2.ManaulOpen := FALSE;
       #DamperController2.ManualClose := TRUE;
   ELSE
       #DamperController2.ManualMode := "MB".Table.HMI_ManualModeOn;
       #DamperController2.ManaulOpen := "MB".Table.HMI_ManualOpenDamper2;
       #DamperController2.ManualClose := NOT "MB".Table.HMI_ManualOpenDamper2;
   END_IF;

   #DamperController2(TankLevel := "MB".Table.RCV2LevelValue,
                      TankLevelSetpoint := ("MB".Table.LevelRCV2Min + ("MB".Table.LevelRCV2Max - "MB".Table.LevelRCV2Min) / 2),
                      TankLevelMin := "MB".Table.LevelRCV2Min,
                      TankLevelMax := "MB".Table.LevelRCV2Max,
                      UsePID := "MB".Table.UsePID,
                      PID_DeadZone := "MB".Table.Damper2_PID_SetpointDeadZone,
                      PID_KP := "MB".Table.Damper2_PID_KP,
                      PID_KI := "MB".Table.Damper2_PID_KI,
                      PID_KD := "MB".Table.Damper2_PID_KD,
                      PID_TI := "MB".Table.Damper2_PID_TI,
                      LimitSwitch0 := "RunClose2",
                      LimitSwitch100 := "RunOpen2",
                      PouseMove := 5,
                      PositionDeadzone := "MB".Table.Damper2_PositionDeadZone,
                      StartAjustment := "Config".HMI_StartAdjustDamper2,
                      CancelAjustment := "Config".HMI_StopAdjustDamper2,
                      ResetPosition := "Config".HMI_ResetPositionDamper2,
                      Open => "OutOpen2",
                      Close => "OutClose2",
                      FullMovingTime := "MB".Table.Damper2_FullMovingTime,
                      SwitchAutoMode := "Damper2_AutoMode");

   "MB".Table.Damper2_Position := #DamperController2.CurrentPosition;
   "MB".Table.Damper2_PositionSetpoint := #DamperController2.PositionSetPoint;
   "MB".Table.Damper2_PID_Setpoint := #DamperController2.TankLevelSetpoint;
   "MB".Table.Damper2_AdjustBusy := #DamperController2.AdjustBusy;
   "MB".Table.Damper2_AdjustError := #DamperController2.AdjustError;
   "MB".Table.Damper2_AdjustDone := WORD_TO_BOOL(#DamperController2.AdjustmentDone);

   "MB".Table."Damper2_Manual/Auto" := "Damper2_AutoMode";

   #DamperController3(TankLevel := "MB".Table.RCV1LevelValue,
                      TankLevelMin := "MB".Table.LevelRCV1Min,
                      TankLevelMax := "MB".Table.LevelRCV1Max,
                      UsePID := FALSE,
                      LimitSwitch0 := "RunClose1",
                      LimitSwitch100 := "RunOpen1",
                      PouseMove := 5,
                      PositionDeadzone := "MB".Table.Damper1_PositionDeadZone,
                      Open => "OsmosOut",
                      FullMovingTime := "MB".Table.Damper1_FullMovingTime,
                      SwitchAutoMode := TRUE);



   IF "MB".Table.RCV1LevelValue < "MB".Table.LevelRCV1Min THEN
       "OsmosAO" := 5520;
   ELSIF "MB".Table.RCV1LevelValue > "MB".Table.LevelRCV1Max THEN
       "OsmosAO" := 27648;
   ELSE
       "OsmosAO" := REAL_TO_INT(("MB".Table.RCV1LevelValue - "MB".Table.LevelRCV1Min) / ("MB".Table.LevelRCV1Max - "MB".Table.LevelRCV1Min) * (27648 - 5520) + 5520);
   END_IF;

   IF "Inputs_DB".ErrorRCV2 THEN
       #DamperController3.ManualMode := TRUE;
       #DamperController3.ManaulOpen := FALSE;
       #DamperController3.ManualClose := TRUE;
   END_IF;



   IF "MB".Table.Damper2_Position > 0 THEN
       "MB".Table."Damper2_Close/Open" := TRUE;
   ELSE
       "MB".Table."Damper2_Close/Open" := FALSE;
   END_IF;
END_FUNCTION_BLOCK

FUNCTION_BLOCK "DamperController"   // FB8, SCL
{ S7_Optimized_Access := 'TRUE' }
VERSION : 0.1
// stored: AutoNumber true, IsIECCheckEnabled false, IsRetainMemResEnabled false, MemoryReserve 100, SetENOAutomatically false, UDAEnableTagReadback false
   VAR_INPUT
      ManualMode : Bool;
      ManaulOpen : Bool;
      ManualClose : Bool;
      TankLevel : Real;
      TankLevelSetpoint : Real;
      TankLevelMin : Real;
      TankLevelMax : Real;
      UsePID : Bool;
      PID_DeadZone : Real;
      PID_KP : Real;
      PID_KI : Real;
      PID_KD : Real;
      PID_TI : Real;
      LimitSwitch0 : Bool;
      LimitSwitch100 : Bool;
      PouseMove : UInt := 10;
      PositionDeadzone : Real := 1.0;
      StartAjustment : Bool;
      CancelAjustment : Bool;
      ResetPosition : Bool;
      SwitchAutoMode : Bool;
   END_VAR
   VAR_OUTPUT
      Open : Bool;
      Close : Bool;
      CurrentPosition : Real;
      PositionError : Bool;
      PositionSetPoint : Real;
      AdjustBusy : Bool;
      AdjustError : Bool;
   END_VAR
   VAR_IN_OUT
      FullMovingTime : Real;
   END_VAR
   VAR
      MoveToLimitSwitch : Bool;
      AdjustmentDone : Word;
      LappedSetpoint : Real;
      isMoving : Bool;
      isAutoMode : Bool;
      isReady : Bool;
      EnablePIDTON { S7_SetPoint := 'True'} : TON_TIME;
      PIDRegulator { S7_SetPoint := 'True'} : "PIDRegulator";
      HystRegulator { S7_SetPoint := 'True'} : "HystRegulator";
      RepositionRTrig { S7_SetPoint := 'True'} : R_TRIG;
      MotorPositionNoFeedback { S7_SetPoint := 'True'} : "MotorPositionNoFeedback";
      MotorController { S7_SetPoint := 'True'} : "MotorControllerSimple";
      RepositionTON { S7_SetPoint := 'True'} : TON_TIME;
      MotorMoverToSwitch { S7_SetPoint := 'True'} : "MotorMoverToSwitch";
      MotorAdjustmentNoFeedback { S7_SetPoint := 'True'} : "MotorAdjustmentNoFeedback";
   END_VAR
   VAR CONSTANT
      LappingZone0 : Real := 1.0;
      LappingZone100 : Real := 2.0;
      EnablePIDTime : Time := T#10s;
   END_VAR
BEGIN
   #isMoving := #Open OR #Close;
   #isAutoMode := NOT #ManualMode;
   #isReady := #isAutoMode;

   #EnablePIDTON(IN:=#UsePID AND #isReady,
                 PT:= #EnablePIDTime);

   #PIDRegulator(Enable:=#EnablePIDTON.Q,
                 Tanklevel:=#TankLevel,
                 TankLevelSetpoint:=#TankLevelSetpoint,
                 KP:=#PID_KP,
                 KI:=#PID_KI,
                 KD:=#PID_KD,
                 TI:=DINT_TO_TIME(REAL_TO_DINT(#PID_TI)*1000),
                 LimitMin:=0,
                 DeadZone := #PID_DeadZone);


   #PositionSetPoint := LIMIT(MN := 0, IN := #PIDRegulator.DamperPosition, MX := 100);

   IF #TankLevel > #TankLevelMax THEN
       #PositionSetPoint := 0;
   END_IF;

   IF #TankLevel < #TankLevelMin THEN
       #PositionSetPoint := 100;
   END_IF;

   #HystRegulator(Enable:=#isAutoMode AND (NOT #UsePID),
                  TankLevel:=#TankLevel,
                  TankLevelMin:=#TankLevelMin,
                  TankLevelMax:=#TankLevelMax);

   #RepositionRTrig(CLK:=#ResetPosition);

   #MotorPositionNoFeedback(Enable:=TRUE,
                            LimitSwitch0:=#LimitSwitch0,
                            LimitSwitch100:=#LimitSwitch100,
                            Invalidate:=#RepositionRTrig.Q,
                            FullMovingTime:=#FullMovingTime,
                            LappingZone:=#PositionDeadzone,
                            Open:=#Open,
                            Close:=#Close,
                            CurrentPosition=>#CurrentPosition,
                            Error=>#PositionError,
                            SwitchAutoMode := #SwitchAutoMode);

   #LappedSetpoint := #PositionSetPoint;
   IF #PositionSetPoint <= #LappingZone0 THEN
       #LappedSetpoint := 0;
   ELSIF #PositionSetPoint >= (100 - #LappingZone100) THEN
       #LappedSetpoint := 100;
   END_IF;

   #MotorController(Enable := #isAutoMode AND #UsePID,
                    CurrentPosition := #CurrentPosition,
                    SetpointPosition := #LappedSetpoint,
                    PositionDeadzone := #PositionDeadzone,
                    MinimalPulse := REAL_TO_DINT(LIMIT(MN := 0.1, IN := #FullMovingTime / 100, MX := 0.5) * 1000),
                    PauseMode := UINT_TO_TIME(IN := #PouseMove) * 1000,
                    isMoving := #isMoving,
                    MoveNow := FALSE,
                    MinReversPause := T#2s,
                    PositionError:=#PositionError);


   #RepositionTON(IN:=TRUE,
                  PT:=T#10s);

   #MotorMoverToSwitch(Enable:=#RepositionTON.Q,
                       Go:= #PositionError,
                       TargetSwitch100:=FALSE,
                       MovePause:=T#5s,
                       isMoving:=#isMoving,
                       LimitSwitch0:=#LimitSwitch0,
                       LimitSwitch100:=#LimitSwitch100);

   #MotorAdjustmentNoFeedback(Enable:=#isAutoMode,
                              Start:=#StartAjustment,
                              Cancel:=#CancelAjustment,
                              AbortTime:=T#120s,
                              MovePause:=T#5s,
                              isMoving:=#isMoving,
                              LimitSwitch0:=#LimitSwitch0,
                              LimitSwitch100:=#LimitSwitch100,
                              Done:=#AdjustmentDone,
                              FullMovingTime:=#FullMovingTime,
                              Busy => #AdjustBusy,
                              Error => #AdjustError);

   IF ("MB".Table.Alarms_NoPowerSupply OR NOT #SwitchAutoMode) THEN
       #Open := FALSE;
       #Close := FALSE;
       RETURN;
   END_IF;

   IF #ManualMode THEN
       #Open := #ManaulOpen;
       #Close := #ManualClose;

   ELSIF #MotorAdjustmentNoFeedback.Busy THEN
       #Open := #MotorAdjustmentNoFeedback.Open;
       #Close := #MotorAdjustmentNoFeedback.Close;

   ELSIF #PositionError THEN
       #Open := #MotorMoverToSwitch.Open;
       #Close := #MotorMoverToSwitch.Close;

   ELSIF #UsePID THEN
       #Open := #MotorController.Open;
       #Close := #MotorController.Close;
   ELSE
       #Open := #HystRegulator.Open;
       #Close := #HystRegulator.Close;
       #PositionSetPoint := #HystRegulator.PositionSetpoint;
   END_IF;
END_FUNCTION_BLOCK

FUNCTION_BLOCK "PIDRegulator"   // FB9, SCL
{ S7_Optimized_Access := 'TRUE' }
VERSION : 0.1
// stored: AutoNumber true, IsIECCheckEnabled false, IsRetainMemResEnabled false, MemoryReserve 100, SetENOAutomatically false, UDAEnableTagReadback false
   VAR_INPUT
      Enable : Bool;
      Tanklevel : Real;
      TankLevelSetpoint : Real;
      KP : Real := 2.0;
      KI : Real := 0.2;
      KD : Real := 0.5;
      TI : Time := T#1s;
      LimitMin : Real := -100.0;
      LimitMax : Real := 100.0;
      DeadZone : Real := 1.0;
   END_VAR
   VAR_OUTPUT
      DamperPosition : Real;
   END_VAR
   VAR
      "e" : Real;
      PValue : Real;
      IValue : Real;
      DValue : Real;
      init : Bool;
      TopLevelSetPoint : Real;
      BottomlevelSetPoint : Real;
      PrevValue : Real;
      TON1 { S7_SetPoint := 'True'} : TON_TIME;
   END_VAR
BEGIN
   IF NOT #Enable THEN
       #init := false;
       #IValue := 0;
       #DValue := 0;
   END_IF;

   IF NOT #init THEN
       #PrevValue := #Tanklevel;
       #init := TRUE;
   END_IF;

   #TopLevelSetPoint := #TankLevelSetpoint + #DeadZone;
   #BottomlevelSetPoint := #TankLevelSetpoint - #DeadZone;

   IF #Tanklevel > #TopLevelSetPoint THEN
       #e := #TopLevelSetPoint - #Tanklevel;
   ELSIF #Tanklevel < #BottomlevelSetPoint THEN
       #e := #BottomlevelSetPoint - #Tanklevel;
   ELSE
       #e := 0;
       #PrevValue := #Tanklevel;
   END_IF;



   #TON1(IN:=TRUE,
         PT:=#TI);



   IF #TON1.Q THEN
       #IValue := #IValue + #e * #KI;
       #IValue := LIMIT(MN := #LimitMin, IN := #IValue, MX := #LimitMax);

       IF #KI <= 0.00001 THEN
           #IValue := 0;
       END_IF;
       #PValue := #e * #KP;
       #DValue := (#Tanklevel - #PrevValue) * #KD;
       #PrevValue := #Tanklevel;
       #DamperPosition := #PValue + #IValue - #DValue;
       RESET_TIMER(#TON1);
   END_IF;
END_FUNCTION_BLOCK

FUNCTION_BLOCK "HystRegulator"   // FB10, SCL
{ S7_Optimized_Access := 'TRUE' }
VERSION : 0.1
// stored: AutoNumber true, IsIECCheckEnabled false, IsRetainMemResEnabled false, MemoryReserve 100, SetENOAutomatically false, UDAEnableTagReadback false
   VAR_INPUT
      Enable { ExternalAccessible := 'False'; ExternalVisible := 'False'; ExternalWritable := 'False'} : Bool;
      TankLevel { ExternalAccessible := 'False'; ExternalVisible := 'False'; ExternalWritable := 'False'} : Real;
      TankLevelMin { ExternalAccessible := 'False'; ExternalVisible := 'False'; ExternalWritable := 'False'} : Real;
      TankLevelMax { ExternalAccessible := 'False'; ExternalVisible := 'False'; ExternalWritable := 'False'} : Real;
   END_VAR
   VAR_OUTPUT
      Open { ExternalAccessible := 'False'; ExternalVisible := 'False'; ExternalWritable := 'False'} : Bool;
      Close { ExternalAccessible := 'False'; ExternalVisible := 'False'; ExternalWritable := 'False'} : Bool;
      PositionSetpoint { ExternalAccessible := 'False'; ExternalVisible := 'False'; ExternalWritable := 'False'} : Real;
   END_VAR
BEGIN
   IF NOT #Enable THEN
       #Open := FALSE;
       #Close := FALSE;
       #PositionSetpoint := 0;
       RETURN;
   END_IF;

   IF #TankLevel <= #TankLevelMin THEN
       #Open := TRUE;
       #Close := FALSE;
       #PositionSetpoint := 100;
   END_IF;

   IF #TankLevel >= #TankLevelMax THEN
       #Open := FALSE;
       #Close := TRUE;
       #PositionSetpoint := 0;
   END_IF;
END_FUNCTION_BLOCK

FUNCTION_BLOCK "MotorPositionNoFeedback"   // FB11, SCL
{ S7_Optimized_Access := 'TRUE' }
VERSION : 0.1
// stored: AutoNumber true, IsIECCheckEnabled false, IsRetainMemResEnabled false, MemoryReserve 100, SetENOAutomatically false, UDAEnableTagReadback false
   VAR_INPUT
      Enable : Bool;
      LimitSwitch0 : Bool;
      LimitSwitch100 : Bool;
      Invalidate : Bool := False;
      FullMovingTime : Real;
      LappingZone : Real := 1.0;
      Open : Bool;
      Close : Bool;
      SwitchAutoMode : Bool;
   END_VAR
   VAR_OUTPUT
      CurrentPosition : Real;
      Error : Bool := FALSE;
   END_VAR
   VAR
      PreviousPosition : Real;
      OnePercentImpulse : Real;
      MovingTimer1 { S7_SetPoint := 'True'} : TON_TIME;
      MovingTimer2 { S7_SetPoint := 'True'} : TON_TIME;
   END_VAR
BEGIN
   #LappingZone := LIMIT(MN := 1.0, IN := #LappingZone, MX := 30.0);

   IF #Enable THEN
       #MovingTimer1(IN:=#Open, PT:= DINT_TO_TIME(REAL_TO_DINT(#FullMovingTime)*1000/100));
       #MovingTimer2(IN:=#Close,PT:= DINT_TO_TIME(REAL_TO_DINT(#FullMovingTime)*1000/100));

       IF #Error = FALSE THEN
           IF #Open AND #MovingTimer1.Q THEN
               #CurrentPosition := #PreviousPosition + 1;
               #CurrentPosition := MIN(IN1 := #CurrentPosition, IN2 := 100-#LappingZone);
               RESET_TIMER(#MovingTimer1);
               #PreviousPosition := #CurrentPosition;
           END_IF;

           IF #Close AND #MovingTimer2.Q THEN
               #CurrentPosition := #PreviousPosition - 1;
               #CurrentPosition := MAX(IN1 := #CurrentPosition, IN2 := #LappingZone);
               RESET_TIMER(#MovingTimer2);
               #PreviousPosition := #CurrentPosition;
           END_IF;
       END_IF;

       IF #LimitSwitch100 THEN
           #CurrentPosition := 100;
           #Error := 0;
           #PreviousPosition := #CurrentPosition;
           RESET_TIMER(#MovingTimer1);
           RESET_TIMER(#MovingTimer2);
       END_IF;

       IF #LimitSwitch0 THEN
           #CurrentPosition := 0;
           #Error := 0;
           #PreviousPosition := #CurrentPosition;
           RESET_TIMER(#MovingTimer1);
           RESET_TIMER(#MovingTimer2);
       END_IF;

       IF #Invalidate THEN
           #CurrentPosition := 0;
           #Error := TRUE;
       END_IF;
   ELSE
       #CurrentPosition := 0;
       #Error := TRUE;
       RESET_TIMER(#MovingTimer1);
       RESET_TIMER(#MovingTimer2);
   END_IF;
END_FUNCTION_BLOCK

FUNCTION_BLOCK "MotorControllerSimple"   // FB12, SCL
{ S7_Optimized_Access := 'TRUE' }
VERSION : 0.1
// stored: AutoNumber true, IsIECCheckEnabled false, IsRetainMemResEnabled false, MemoryReserve 100, SetENOAutomatically false, UDAEnableTagReadback false
   VAR_INPUT
      Enable : Bool;
      CurrentPosition : Real;
      SetpointPosition : Real;
      PositionDeadzone : Real := 2.0;
      MinimalPulse : Time;
      PauseMode : Time := T#10s;
      isMoving : Bool;
      MoveNow : Bool;
      MinReversPause : Time := T#1s;
      PositionError : Bool;
   END_VAR
   VAR_OUTPUT
      Open : Bool;
      Close : Bool;
   END_VAR
   VAR
      Opening : Bool;
      Closing : Bool;
      MovingTOF { S7_SetPoint := 'True'} : TOF_TIME;
      OpeningTOF { S7_SetPoint := 'True'} : TOF_TIME;
      ClosingTOF { S7_SetPoint := 'True'} : TOF_TIME;
      TON1 { S7_SetPoint := 'True'} : TON_TIME;
      TON2 { S7_SetPoint := 'True'} : TON_TIME;
   END_VAR
BEGIN
   #MovingTOF(IN:=(#isMoving OR #Open OR #Close),
              PT:=#PauseMode);
   #OpeningTOF(IN:=#Open,
               PT:=#MinReversPause);
   #ClosingTOF(IN:=#Close,
               PT:=#MinReversPause);

   IF #Enable AND NOT #PositionError THEN
       IF (NOT #MovingTOF.Q) OR #MoveNow THEN
           IF #CurrentPosition < #SetpointPosition - #PositionDeadzone THEN
               #Opening := TRUE;
               #Closing := FALSE;
           END_IF;
           IF #CurrentPosition > #SetpointPosition + #PositionDeadzone THEN
               #Opening := FALSE;
               #Closing := TRUE;
           END_IF;
           IF #SetpointPosition = 0 THEN
               #Opening := FALSE;
               #Closing := TRUE;
           END_IF;
           IF #SetpointPosition = 100 THEN
               #Opening := TRUE;
               #Closing := FALSE;
           END_IF;

       END_IF;

       IF #Opening AND #CurrentPosition >= #SetpointPosition - 0.1 THEN
           #Opening := FALSE;
       END_IF;
       IF #Closing AND #CurrentPosition <= #SetpointPosition + 0.1 THEN
           #Closing := FALSE;
       END_IF;

       IF #Opening AND (NOT #ClosingTOF.Q) THEN
           #Open := TRUE;
       ELSIF (NOT #Opening) AND #TON1.Q THEN
           #Open := FALSE;
       END_IF;

       #TON1(IN:=#Open,
             PT:=#MinimalPulse);

       IF #Closing AND (NOT #OpeningTOF.Q) THEN
           #Close := TRUE;
       ELSIF (NOT #Closing) AND #TON2.Q THEN
           #Close := FALSE;
       END_IF;

       #TON2(IN:=#Close,
             PT:=#MinimalPulse);
   ELSE
       #Open := FALSE;
       #Close := FALSE;
       #Opening := FALSE;
       #Closing := FALSE;
       RESET_TIMER(#TON1);
       RESET_TIMER(#TON2);
   END_IF;
END_FUNCTION_BLOCK

FUNCTION_BLOCK "MotorMoverToSwitch"   // FB13, SCL
{ S7_Optimized_Access := 'TRUE' }
VERSION : 0.1
// stored: AutoNumber true, IsIECCheckEnabled false, IsRetainMemResEnabled false, MemoryReserve 100, SetENOAutomatically false, UDAEnableTagReadback false
   VAR_INPUT
      Enable : Bool;
      Go : Bool;
      TargetSwitch100 : Bool := True;
      MovePause : Time := T#10s;
      isMoving : Bool;
      LimitSwitch0 : Bool;
      LimitSwitch100 : Bool;
   END_VAR
   VAR_OUTPUT
      Open : Bool;
      Close : Bool;
   END_VAR
   VAR
      GoTo0 : Bool;
      GoTo100 : Bool;
      MovingTOF { S7_SetPoint := 'True'} : TOF_TIME;
   END_VAR
BEGIN
   #MovingTOF(IN:=#isMoving,
              PT:=#MovePause);

   IF #Enable THEN
       IF (NOT #MovingTOF.Q) AND #TargetSwitch100 AND #Go THEN
           #GoTo100 := TRUE;
       END_IF;
       IF #LimitSwitch100 OR (NOT #TargetSwitch100) OR (NOT #Go) THEN
           #GoTo100 := FALSE;
       END_IF;

       IF (NOT #MovingTOF.Q) AND (NOT #TargetSwitch100) AND #Go THEN
           #GoTo0 := #Go;
       END_IF;
       IF #LimitSwitch0 OR #TargetSwitch100 OR (NOT #Go) THEN
           #GoTo0 := FALSE;
       END_IF;

       IF #GoTo100 THEN
           #Open := TRUE;
           #Close := FALSE;
       ELSIF #GoTo0 THEN
           #Open := FALSE;
           #Close := TRUE;
       ELSE
           #Open := FALSE;
           #Close := FALSE;
       END_IF;
   ELSE
       #Open := FALSE;
       #Close := FALSE;
       #GoTo0 := FALSE;
       #GoTo100 := FALSE;
   END_IF;
END_FUNCTION_BLOCK

FUNCTION_BLOCK "MotorAdjustmentNoFeedback"   // FB14, SCL
{ S7_Optimized_Access := 'TRUE' }
VERSION : 0.1
// stored: AutoNumber true, IsIECCheckEnabled false, IsRetainMemResEnabled false, MemoryReserve 100, SetENOAutomatically false, UDAEnableTagReadback false
   VAR_INPUT
      Enable : Bool;
      Start : Bool;
      Cancel : Bool;
      AbortTime : Time := T#120s;
      MovePause : Time := T#10s;
      isMoving : Bool;
      LimitSwitch0 : Bool;
      LimitSwitch100 : Bool;
   END_VAR
   VAR_OUTPUT
      Busy : Bool;
      Error : Bool;
      Open : Bool;
      Close : Bool;
   END_VAR
   VAR_IN_OUT
      Done : Word;
      FullMovingTime : Real;
   END_VAR
   VAR
      "step" : Word;
      StartRTrig { S7_SetPoint := 'True'} : R_TRIG;
      CancelRTrig { S7_SetPoint := 'True'} : R_TRIG;
      MovingTOF { S7_SetPoint := 'True'} : TOF_TIME;
      MovingTON { S7_SetPoint := 'True'} : TON_TIME;
      PauseTON { S7_SetPoint := 'True'} : TON_TIME;
   END_VAR
BEGIN
   #StartRTrig(CLK:=#Start);
   IF #StartRTrig.Q AND #step = 0 THEN
       #step := 1;
   END_IF;

   #CancelRTrig(CLK:=#Cancel);

   IF #CancelRTrig.Q THEN
       #step := 0;
       #Error := FALSE;
   END_IF;

   IF NOT #Enable THEN
       #step := 0;
   END_IF;

   #MovingTOF(IN:=#isMoving,
              PT:=#MovePause);


   CASE #step OF
       1:
           #Busy := TRUE;
           #Done := 0;
           #Error := FALSE;
           IF NOT #MovingTOF.Q THEN
               #step += 1;
           END_IF;

       2:
           #Open := FALSE;
           #Close := TRUE;
           #step += 1;
       3:
           #MovingTON(IN := TRUE,
                      PT := #AbortTime);
           IF #LimitSwitch0 THEN
               #step += 1;
               RESET_TIMER(#MovingTON);
           END_IF;
           IF #MovingTON.Q THEN
               #Error := TRUE;
               RESET_TIMER(#MovingTON);
               #step := 10;
           END_IF;
       4:
           #Open := FALSE;
           #Close := FALSE;
           #PauseTON(IN := TRUE,
                     PT := #MovePause);
           IF #PauseTON.Q THEN
               RESET_TIMER(#PauseTON);
               #step += 1;
           END_IF;
       5:
           #Open := True;
           #Close := FALSE;
           #step += 1;
       6:
           #MovingTON(IN := TRUE,
                      PT := #AbortTime);
           #step += 1;
       7:
           IF #LimitSwitch100 THEN
               #step += 1;
           END_IF;
           IF #MovingTON.Q THEN
               #Error := True;
               RESET_TIMER(#MovingTON);
               #step := 10;
           END_IF;
       8:
           #FullMovingTime := DINT_TO_REAL(IN := #MovingTON.ET) / 1000;
           RESET_TIMER(#MovingTON);
           #step += 1;
       9:
           #Open := FALSE;
           #Close := FALSE;
           #PauseTON(IN := TRUE,
                     PT := #MovePause);
           IF #PauseTON.Q THEN
               #step += 1;
           END_IF;
       10:
           #Busy := FALSE;
           #Done := BOOL_TO_WORD(NOT #Error);
           #step := 0;  
       ELSE
           #step := 0;
           #Open := FALSE;
           #Close := FALSE;
           #Busy := FALSE;
           RESET_TIMER(#MovingTON);
           RESET_TIMER(#PauseTON);
   END_CASE;
END_FUNCTION_BLOCK

FUNCTION_BLOCK "Weighting"   // FB18, SCL
{ S7_Optimized_Access := 'FALSE' }
VERSION : 0.1
// stored: AutoNumber true, IsIECCheckEnabled false, SetENOAutomatically false, UDAEnableTagReadback false
   VAR DB_SPECIFIC
      buffer1 { S7_SetPoint := 'True'} : Array[0..1] of Word;
      buffer2 : Array[0..1] of Word;
      Enable { S7_SetPoint := 'True'} : Bool;
      ManualValueProvided1 : Bool;
      ManualValueProvided2 : Bool;
      ManualValue1 : Real;
      ManualValue2 : Real;
   END_VAR
   VAR
      WeightHandlers : Array[0..1] of "WeightHandler";
      TankWeigher1 { S7_SetPoint := 'True'} : "TankWeigher";
   END_VAR
   VAR DB_SPECIFIC
      RetainData : "WeightRetainData";
      TimeNow { S7_SetPoint := 'True'} : DTL;
   END_VAR
   VAR_TEMP
      Temp1 : DWord;
      Temp2 : DWord;
      Ret : Int;
   END_VAR
   VAR CONSTANT
      CLOR_DENSITY : Real := 1.2;
   END_VAR
BEGIN
   #Enable := "MB".Table.WeightingEnable;

   "ModbusLoad"(REQ :="FirstScan",
               PORT := "Local~CM_1241_(RS422_485)_1",
               BAUD := 9600,
               PARITY := 0,
               RESP_TO := 100,
               MB_DB := "ModbusMaster");

   "ModbusMaster"(REQ := "ModbusLoad".DONE,
                 MB_ADDR := 16,
                 MODE := 0,
                 DATA_ADDR := 40063,
                 DATA_LEN := 2,
                 DATA_PTR := "MB".Table.SensorWeightVoltage1);

   "ModbusMaster"(REQ := "ModbusLoad".DONE,
                 MB_ADDR := 17,
                 MODE := 0,
                 DATA_ADDR := 40063,
                 DATA_LEN := 2,
                 DATA_PTR := "MB".Table.SensorWeightVoltage2);

   "ModbusMaster"(REQ := "ModbusLoad".DONE,
                 MB_ADDR := 18,
                 MODE := 0,
                 DATA_ADDR := 40005,
                 DATA_LEN := 2,
                 DATA_PTR := "MB".Table.WaterTemperature);


   IF NOT #Enable THEN
       IF "MB".Table.Weighting_SaveManualValue THEN
           IF "MB".Table.Weighting_ManualValue1 <> 0 THEN
               #ManualValueProvided1 := TRUE;
               #ManualValue1 := "MB".Table.Weighting_ManualValue1 * #CLOR_DENSITY;
           END_IF;
           IF "MB".Table.Weighting_ManualValue2 <> 0 THEN
               #ManualValueProvided2 := TRUE;
               #ManualValue2 := "MB".Table.Weighting_ManualValue1 * #CLOR_DENSITY;
           END_IF;
       END_IF;
   ELSE
       #ManualValueProvided1 := FALSE;
       #ManualValue1 := 0;
       #ManualValueProvided2 := FALSE;
       #ManualValue1 := 0;
   END_IF;

   IF "MB".Table.Weighting_SaveManualValue THEN
       "MB".Table.Weighting_SaveManualValue := FALSE;
   END_IF;



   #WeightHandlers[0](
                      Value := "MB".Table.SensorWeightVoltage1,
                      ValueMin := "MB".Table.WeightVoltageMin1,
                      ValueMax := "MB".Table.WeightVoltageMax1,
                      ValueOffset := "MB".Table.WeightValueOffset1,
                      OutputMin := "MB".Table.WeightValueMin1,
                      OutputMax := "MB".Table.WeightValueMax1,
                      Output => "MB".Table.WeightValue1);

   #WeightHandlers[1](
                      Value := "MB".Table.SensorWeightVoltage2,
                      ValueMin := "MB".Table.WeightVoltageMin2,
                      ValueMax := "MB".Table.WeightVoltageMax2,
                      ValueOffset := "MB".Table.WeightValueOffset2,
                      OutputMin := "MB".Table.WeightValueMin2,
                      OutputMax := "MB".Table.WeightValueMax2,
                      Output => "MB".Table.WeightValue2);

   #Ret := RD_SYS_T(#TimeNow);

   #TankWeigher1(WeightDelay:="MB".Table.WeightingDelay*1000,
                 WeightDeadZone:="MB".Table.WeightingDeadZone,
                 DayTour:="MB".Table.CycleDay,
                 CalendarMonth := #TimeNow.MONTH,
                 CalendarDay := #TimeNow.DAY,
                 ref_RetainData:=#RetainData
   );

   IF #ManualValueProvided1 THEN
       "MB".Table.WeightValue1 := #ManualValue1;
   END_IF;

   IF #ManualValueProvided2 THEN
       "MB".Table.WeightValue2 := #ManualValue2;
   END_IF;

   "MB".Table.WeightValue1Liters := "MB".Table.WeightValue1/ #CLOR_DENSITY;
   "MB".Table.WeightValue2Liters := "MB".Table.WeightValue2 / #CLOR_DENSITY;

   "MB".Table.WeightingStat_CalendarDay := #RetainData.ArrayCalendarDay;
   "MB".Table.WeightingStat_CalendarMonth := #RetainData.ArrayCalendarMonth;
   "MB".Table.WeightingStat_DayCycle := #RetainData.ArrayDayTour;
   "MB".Table.WeightingStat_Counsumed1 := #RetainData.ArrayConsumedFeed1;
   "MB".Table.WeightingStat_Load1 := #RetainData.ArrayLoadedFeed1;
   "MB".Table.WeightingStat_Counsumed2 := #RetainData.ArrayConsumedFeed2;
   "MB".Table.WeightingStat_Load2 := #RetainData.ArrayLoadedFeed2;
   "MB".Table.WeightSensor1Error := #WeightHandlers[0].Error;
   "MB".Table.WeightSensor2Error := #WeightHandlers[1].Error;
END_FUNCTION_BLOCK

FUNCTION_BLOCK "WeightHandler"   // FB20, SCL
{ S7_Optimized_Access := 'TRUE' }
VERSION : 0.1
// stored: AutoNumber true, IsIECCheckEnabled false, IsRetainMemResEnabled false, MemoryReserve 100, SetENOAutomatically false, UDAEnableTagReadback false
   VAR_INPUT
      ValueMin : Real;
      ValueMax : Real;
      OutputMin : Real;
      OutputMax : Real;
      ValueOffset : Real;
      Value : Real;
   END_VAR
   VAR_OUTPUT
      Output : Real;
      Error : Bool;
   END_VAR
   VAR
      ConvertedValue : Real;
      TON1 { S7_SetPoint := 'True'} : TON_TIME;
   END_VAR
BEGIN
   #Error := FALSE;



   #ConvertedValue := (#Value - #ValueMin) / (#ValueMax - #ValueMin) * (#OutputMax - #OutputMin) + #OutputMin;
   #Output := #ConvertedValue + #ValueOffset;

   #TON1(IN := #ConvertedValue < 0.1,
         PT := T#60s,
         Q => #Error);

   IF #Output < 0 THEN
       #Output := 0;
   END_IF;
END_FUNCTION_BLOCK

FUNCTION_BLOCK "TankWeigher"   // FB25, SCL
{ S7_Optimized_Access := 'TRUE' }
VERSION : 0.1
// stored: AutoNumber true, IsIECCheckEnabled false, IsRetainMemResEnabled false, MemoryReserve 100, SetENOAutomatically false, UDAEnableTagReadback false
   VAR_INPUT
      WeightDelay : Time := T#30s;
      WeightDeadZone : Real := 0.1;
      DayTour : Int;
      CalendarDay : UInt;
      CalendarMonth : UInt;
   END_VAR
   VAR_OUTPUT
      IsWeightMessured : Bool;
      IsFeedLoaded : Bool;
      IsFeedConsumed : Bool;
   END_VAR
   VAR_IN_OUT
      ref_RetainData : "WeightRetainData";
   END_VAR
   VAR
      TankDetector1 { S7_SetPoint := 'True'} : "TankDetector";
      TankRegistrator1 { S7_SetPoint := 'True'} : "TankRegistrator";
      TankDetector2 { S7_SetPoint := 'True'} : "TankDetector";
   END_VAR
BEGIN
   #TankDetector1(WeightValue:="MB".Table.WeightValue1,
                  WeightDelay:=#WeightDelay,
                  WeightError:=false,
                  DeadZone:=#WeightDeadZone,
                  IsWeightMeasured=>#IsWeightMessured,
                  IsFeedLoaded=>#IsFeedLoaded,
                  IsFeedConsumed=>#IsFeedConsumed,
                  Ref_ConsumedFeed:=#ref_RetainData.ConsumedFeed1,
                  Ref_LoadedFeed:=#ref_RetainData.LoadedFeed1,
                  Ref_PreviousWeight:=#ref_RetainData.PreviousWeight1);

   #TankDetector2(WeightValue := "MB".Table.WeightValue2,
                  WeightDelay := #WeightDelay,
                  WeightError := false,
                  DeadZone := #WeightDeadZone,
                  IsWeightMeasured => #IsWeightMessured,
                  IsFeedLoaded => #IsFeedLoaded,
                  IsFeedConsumed => #IsFeedConsumed,
                  Ref_ConsumedFeed := #ref_RetainData.ConsumedFeed2,
                  Ref_LoadedFeed := #ref_RetainData.LoadedFeed2,
                  Ref_PreviousWeight := #ref_RetainData.PreviousWeight2);

   #TankRegistrator1(CurrentConsumedFeed1:=#ref_RetainData.ConsumedFeed1,
                     CurrentConsumedFeed2:=#ref_RetainData.ConsumedFeed2,
                     CurrentLoadedFeed1:=#ref_RetainData.LoadedFeed1,
                     CurrentLoadedFeed2:=#ref_RetainData.LoadedFeed2,
                     DayTour:=#DayTour,
                     CalendarDay:=#CalendarDay,
                     CalendarMonth:=#CalendarMonth,
                     ref_RetainData:=#ref_RetainData);


   IF #TankRegistrator1.ResetCounters THEN
       #TankDetector1.Ref_ConsumedFeed := 0;
       #TankDetector1.Ref_LoadedFeed := 0;
       #TankDetector1.Ref_PreviousWeight := 0;
       #TankDetector2.Ref_ConsumedFeed := 0;
       #TankDetector2.Ref_LoadedFeed := 0;
       #TankDetector2.Ref_PreviousWeight := 0;
   END_IF;
END_FUNCTION_BLOCK

FUNCTION_BLOCK "TankDetector"   // FB23, SCL
{ S7_Optimized_Access := 'TRUE' }
VERSION : 0.1
// stored: AutoNumber true, IsIECCheckEnabled false, IsRetainMemResEnabled false, MemoryReserve 100, SetENOAutomatically false, UDAEnableTagReadback false
   VAR_INPUT
      WeightValue : Real;
      WeightDelay : Time := T#30s;
      WeightError : Bool;
      DeadZone : Real := 0.1;
   END_VAR
   VAR_OUTPUT
      IsWeightMeasured : Bool;
      IsFeedLoaded : Bool;
      IsFeedConsumed : Bool;
      MeasuredWeight : Real;
   END_VAR
   VAR_IN_OUT
      Ref_ConsumedFeed : Real;
      Ref_LoadedFeed : Real;
      Ref_PreviousWeight : Real;
   END_VAR
   VAR
      PreviousWeight1 : Real;
      PreviousWeight2 : Real;
      TON1 { S7_SetPoint := 'True'} : TON_TIME;
      TON2 { S7_SetPoint := 'True'} : TON_TIME;
   END_VAR
BEGIN
   IF #WeightError THEN
       #IsWeightMeasured := FALSE;
       #MeasuredWeight := 0;
       RESET_TIMER(#TON1);
       RESET_TIMER(#TON2);
       RETURN;
   END_IF;

   #IsWeightMeasured := FALSE;
   #IsFeedLoaded := FALSE;
   #IsFeedConsumed := FALSE;

   IF ABS(#WeightValue - #Ref_PreviousWeight) > #DeadZone THEN
       IF #WeightValue > #Ref_PreviousWeight THEN
           #TON2(IN := TRUE,
                 PT := #WeightDelay);
           IF #TON2.Q THEN
               #IsWeightMeasured := TRUE;
               #IsFeedLoaded := TRUE;
               #MeasuredWeight := #WeightValue - #Ref_PreviousWeight;
               #Ref_LoadedFeed := #Ref_LoadedFeed + (#WeightValue - #Ref_PreviousWeight);
               #Ref_PreviousWeight := #WeightValue;
               RESET_TIMER(#TON2);
           END_IF;

           IF ABS(#WeightValue - #PreviousWeight2) > #DeadZone THEN
               RESET_TIMER(#TON2);
               #PreviousWeight2 := #WeightValue;
           END_IF;

           RESET_TIMER(#TON1);
           #PreviousWeight1 := 0;

       ELSIF #WeightValue < #Ref_PreviousWeight THEN
           #TON1(IN := TRUE,
                 PT := #WeightDelay);
           IF #TON1.Q THEN
               #IsWeightMeasured := TRUE;
               #IsFeedConsumed := TRUE;
               #MeasuredWeight := #WeightValue - #Ref_PreviousWeight;
               #Ref_ConsumedFeed := #Ref_ConsumedFeed + (#Ref_PreviousWeight - #WeightValue);
               #Ref_PreviousWeight := #WeightValue;
               RESET_TIMER(#TON1);
           END_IF;

           IF ABS(#WeightValue - #PreviousWeight1) > #DeadZone THEN
               RESET_TIMER(#TON1);
               #PreviousWeight1 := #WeightValue;
           END_IF;

           RESET_TIMER(#TON2);
           #PreviousWeight2 := 0;
       END_IF;

   ELSE
       RESET_TIMER(#TON1);
       RESET_TIMER(#TON2);
       #PreviousWeight1 := 0;
       #PreviousWeight2 := 0;
   END_IF;
END_FUNCTION_BLOCK

FUNCTION_BLOCK "TankRegistrator"   // FB24, SCL
{ S7_Optimized_Access := 'TRUE' }
VERSION : 0.1
// stored: AutoNumber true, IsIECCheckEnabled false, IsRetainMemResEnabled false, MemoryReserve 100, SetENOAutomatically false, UDAEnableTagReadback false
   VAR_INPUT
      CurrentConsumedFeed1 : Real;
      CurrentConsumedFeed2 : Real;
      CurrentLoadedFeed1 : Real;
      CurrentLoadedFeed2 : Real;
      DayTour : Int;
      CalendarDay : UInt;
      CalendarMonth : UInt;
   END_VAR
   VAR_OUTPUT
      ResetCounters : Bool;
   END_VAR
   VAR_IN_OUT
      ref_RetainData : "WeightRetainData";
   END_VAR
   VAR
      i : Int;
   END_VAR
   VAR CONSTANT
      c_ARRAY_SIZE : Int := 30;
   END_VAR
BEGIN

   IF #ref_RetainData.PreviousDayTour <> #DayTour THEN
       FOR #i := 0 TO (#c_ARRAY_SIZE - 2) DO
           #ref_RetainData.ArrayConsumedFeed1[c_ARRAY_SIZE - #i] := #ref_RetainData.ArrayConsumedFeed1[c_ARRAY_SIZE - #i - 1];
           #ref_RetainData.ArrayLoadedFeed1[c_ARRAY_SIZE - #i] := #ref_RetainData.ArrayLoadedFeed1[c_ARRAY_SIZE - #i - 1];
           #ref_RetainData.ArrayConsumedFeed2[c_ARRAY_SIZE - #i] := #ref_RetainData.ArrayConsumedFeed2[c_ARRAY_SIZE - #i - 1];
           #ref_RetainData.ArrayLoadedFeed2[c_ARRAY_SIZE - #i] := #ref_RetainData.ArrayLoadedFeed2[c_ARRAY_SIZE - #i - 1];
           #ref_RetainData.ArrayDayTour[c_ARRAY_SIZE - #i] := #ref_RetainData.ArrayDayTour[c_ARRAY_SIZE - #i - 1];
           #ref_RetainData.ArrayCalendarDay[c_ARRAY_SIZE - #i] := #ref_RetainData.ArrayCalendarDay[c_ARRAY_SIZE - #i - 1];
           #ref_RetainData.ArrayCalendarMonth[c_ARRAY_SIZE - #i] := #ref_RetainData.ArrayCalendarMonth[c_ARRAY_SIZE - #i - 1];
       END_FOR;
       #ref_RetainData.PreviousDayTour := #DayTour;
       #ResetCounters := TRUE;
   ELSE
       #ResetCounters := FALSE;
   END_IF;

       #ref_RetainData.ArrayConsumedFeed1[1] := #CurrentConsumedFeed1;
       #ref_RetainData.ArrayLoadedFeed1[1] := #CurrentLoadedFeed1;
       #ref_RetainData.ArrayConsumedFeed2[1] := #CurrentConsumedFeed2;
       #ref_RetainData.ArrayLoadedFeed2[1] := #CurrentLoadedFeed2;
       #ref_RetainData.ArrayDayTour[1] := #DayTour;
       #ref_RetainData.ArrayCalendarDay[1] := #CalendarDay;
       #ref_RetainData.ArrayCalendarMonth[1] := #CalendarMonth;
END_FUNCTION_BLOCK

FUNCTION_BLOCK "MBServer"   // FB19, SCL
{ S7_Optimized_Access := 'TRUE' }
VERSION : 0.1
// stored: AutoNumber true, IsIECCheckEnabled false, IsRetainMemResEnabled false, MemoryReserve 100, SetENOAutomatically false, UDAEnableTagReadback false
BEGIN
   "MB_SERVER_DB"(DISCONNECT:=FALSE,
                  NDR=>"MB_Config".NDR,
                  DR=>"MB_Config".DR,
                  ERROR=>"MB_Config".ERROR,
                  MB_HOLD_REG:="MB".Table,
                  CONNECT:="MB_Config".CONNECT);
END_FUNCTION_BLOCK

FUNCTION_BLOCK "ModbusClO2"   // FB26, SCL
{ S7_Optimized_Access := 'FALSE' }
VERSION : 0.1
// stored: AutoNumber true, IsIECCheckEnabled false, SetENOAutomatically false, UDAEnableTagReadback false
   VAR DB_SPECIFIC
      ProportionalDosingExternal { S7_SetPoint := 'True'} : DWord;
      AbsoluteDosing : DWord;
      SystemProductivity : DWord;
      Pressure : Word;
      Doser1Productivity : Word;
      Doser2Productivity : Word;
   END_VAR
BEGIN
   "ModbusMaster"(REQ := "ModbusLoad".DONE,
                        MB_ADDR := 1,
                        MODE := 0,
                        DATA_ADDR := 40014,
                        DATA_LEN := 1,
                        DATA_PTR := "MB".Table.ClO2.WorkMode); //OK

   "ModbusMaster"(REQ := "ModbusLoad".DONE,
         MB_ADDR := 1,
         MODE := 0,
         DATA_ADDR := 40015,
         DATA_LEN := 1,
         DATA_PTR := #Doser1Productivity);


   "MB".Table.ClO2.Doser1Productivity := #Doser1Productivity / 100;

   "ModbusMaster"(REQ := "ModbusLoad".DONE,
                 MB_ADDR := 1,
                 MODE := 0,
                 DATA_ADDR := 40016,
                 DATA_LEN := 1,
                 DATA_PTR := #Doser2Productivity);

   "MB".Table.ClO2.Doser2Productivity := #Doser2Productivity / 100;

   "ModbusMaster"(REQ := "ModbusLoad".DONE,
                 MB_ADDR := 1,
                 MODE := 0,
                 DATA_ADDR := 40020,
                 DATA_LEN := 1,
                 DATA_PTR := #Pressure);


   "MB".Table.ClO2.Pressure := #Pressure / 100;

   "ModbusMaster"(REQ := "ModbusLoad".DONE,
                 MB_ADDR := 1,
                 MODE := 0,
                 DATA_ADDR := 40025,
                 DATA_LEN := 2,
                 DATA_PTR := #SystemProductivity);

   "MB".Table.ClO2.SystemProductivity := DWORD_TO_REAL(ROL(IN := #SystemProductivity, N := 16));

   "ModbusMaster"(REQ := "ModbusLoad".DONE,
                 MB_ADDR := 1,
                 MODE := 0,
                 DATA_ADDR := 40010,
                 DATA_LEN := 1,
                 DATA_PTR := "MB".Table.ClO2.ChooseDosing); //OK

   "ModbusMaster"(REQ := "ModbusLoad".DONE,
                 MB_ADDR := 1,
                 MODE := 0,
                 DATA_ADDR := 40012,
                 DATA_LEN := 1,
                 DATA_PTR := "MB".Table.ClO2.DosersActive); //OK

   "ModbusMaster"(REQ := "ModbusLoad".DONE,
                 MB_ADDR := 1,
                 MODE := 0,
                 DATA_ADDR := 40051,
                 DATA_LEN := 2,
                 DATA_PTR := #AbsoluteDosing);

   "MB".Table.ClO2.AbsoluteDosing := DWORD_TO_REAL(ROL(IN := #AbsoluteDosing, N := 16));

   "ModbusMaster"(REQ := "ModbusLoad".DONE,
                 MB_ADDR := 1,
                 MODE := 0,
                 DATA_ADDR := 40055,
                 DATA_LEN := 2,
                 DATA_PTR := #ProportionalDosingExternal);

   "MB".Table.ClO2.ProportionalDosingExternal := DWORD_TO_REAL(ROL(IN := #ProportionalDosingExternal, N := 16));


   "ModbusMaster"(REQ := "ModbusLoad".DONE,
                 MB_ADDR := 1,
                 MODE := 0,
                 DATA_ADDR := 40011,
                 DATA_LEN := 1,
                 DATA_PTR := "MB".Table.ClO2.Alarms); //OK
END_FUNCTION_BLOCK

FUNCTION_BLOCK "ChlorMode"   // FB5, SCL
{ S7_Optimized_Access := 'TRUE' }
VERSION : 0.1
// stored: AutoNumber true, IsIECCheckEnabled false, IsRetainMemResEnabled false, MemoryReserve 100, SetENOAutomatically false, UDAEnableTagReadback false
   VAR
      WaterLevel : Real;
      WaterPulse_RT { S7_SetPoint := 'True'} : R_TRIG;
      PulseSetpoint { S7_SetPoint := 'True'} : Real;
      FreqTON { S7_SetPoint := 'True'} : TON_TIME;
      LevelAlarm { S7_SetPoint := 'True'} : Bool;
      DelayTOF { S7_SetPoint := 'True'} : TOF_TIME;
      PulseGen { S7_SetPoint := 'True'} : TP_TIME;
      DoserValue { S7_SetPoint := 'True'} : Real := 0.0;
      DoserPreValue : Real;
      StopTrig { S7_SetPoint := 'True'} : R_TRIG;
      StartTrig { S7_SetPoint := 'True'} : R_TRIG;
      ChlorMeasurment { S7_SetPoint := 'True'} : "ChlorMeasurment";
      BlockDosing { S7_SetPoint := 'True'} : Bool;
      EnableMeasureTime : Real;
      BlockDosingTime : Real;
   END_VAR
   VAR CONSTANT
      Freq : UDInt := 10;
   END_VAR
BEGIN
   "DoserOut" := FALSE;

   //#WaterPulse_RT(CLK := "WaterCounterOutPulse");
   #ChlorMeasurment(blockDosing=>#BlockDosing);

   "Config".DiOxydeDosing := REAL_TO_DWORD("MB".Table.ChlorationParams.ActualDose);
   "Config".DiOxydeDosing := ROL(IN := "Config".DiOxydeDosing, N := 16);
   "ModbusMaster"(REQ := "ModbusLoad".DONE,
                  MB_ADDR := 1,
                  MODE := 1,
                  DATA_ADDR := 40055,
                  DATA_LEN := 2,
                  DATA_PTR := "Config".DiOxydeDosing);

   IF NOT "MB".Table.HMI_ChlorModeOn OR NOT "MB".Table.Chlor_AutoMode THEN
       "MB".Table.ChlorationParams.ActualDose := 0;

   END_IF;

   IF "MB".Table.HMI_Chlor_ChooseTank = 0 THEN
       #LevelAlarm := "MB".Table.Alarms_RCV1Min OR "MB".Table.Alarms_RCV1Max;
   END_IF;

   IF "MB".Table.HMI_Chlor_ChooseTank = 1 THEN
       #LevelAlarm := "MB".Table.Alarms_RCV2Min OR "MB".Table.Alarms_RCV2Max;
   END_IF;

   "MB".Table.DoserNotWork := (
       #LevelAlarm OR
       "MB".Table.Alarms_ChlorLargeConsumption OR
       #BlockDosing OR
       "MB".Table.CriticalMeasureON
       );

   REGION ChlorationAlgorithm
       // Statement section REGION
       #StartTrig(CLK := "MB".Table.Chlor_StartManual);
       IF #StartTrig.Q THEN
           #DoserValue := 0;
           #DoserPreValue := "MB".Table.Doser1_DailyValue;
       END_IF;

       IF "MB".Table.Chlor_AutoMode THEN
           #FreqTON(IN := #PulseSetpoint > 0,
                    PT := UDINT_TO_DINT(500));
           IF "MB".Table.HMI_ChlorModeOn THEN
               IF "Config".WaterPulseDuble THEN
                   "Config".WaterPulseDuble := FALSE;
                   #PulseSetpoint += "MB".Table.ChlorationParams.ActualDose / "MB".Table.Chlor_PulseWeight_1 * "MB".Table.WaterCounterOut_PulseValue;
               END_IF;



           END_IF;
           IF #FreqTON.Q THEN
               IF #PulseSetpoint >= 0 THEN
                   #PulseGen(IN := #FreqTON.Q,
                             PT := UDINT_TO_DINT(250));
                   #PulseSetpoint -= 1;
               END_IF;
               RESET_TIMER(#FreqTON);
           END_IF;

           IF #PulseGen.Q THEN
               "DoserOut" := True;
               RESET_TIMER(#PulseGen);
           END_IF;
       ELSIF NOT "MB".Table.Chlor_AutoMode AND "MB".Table.Chlor_StartManual THEN
           #StopTrig(CLK := #DoserValue > "MB".Table.Chlor_ManualSetpoint_1 * 1000);
           IF #StopTrig.Q THEN
               "MB".Table.HMI_WeightAlarmReset := 1;
               "MB".Table.Chlor_StartManual := 0;
               RETURN;
           END_IF;

           #DoserValue := "MB".Table.Doser1_DailyValue - #DoserPreValue;
           #FreqTON(IN := #DoserValue < "MB".Table.Chlor_ManualSetpoint_1 * 1000,
                    PT := UDINT_TO_DINT(500));
           IF #FreqTON.Q THEN
               #PulseGen(IN := #FreqTON.Q,
                         PT := UDINT_TO_DINT(250));
               RESET_TIMER(#FreqTON);
           END_IF;

           IF #PulseGen.Q THEN
               IF #DoserValue < "MB".Table.Chlor_ManualSetpoint_1 * 1000 THEN
                   "DoserOut" := True;
                   RESET_TIMER(#PulseGen);
               END_IF;
           END_IF;
       END_IF;
   END_REGION



   IF "MB".Table.DoserNotWork AND "MB".Table.Chlor_AutoMode THEN
       #PulseSetpoint := 0;
       "MB".Table.ChlorationParams.ActualDose := 0;
   END_IF;
END_FUNCTION_BLOCK

FUNCTION_BLOCK "ChlorMeasurment"   // FB21, SCL
{ S7_Optimized_Access := 'TRUE' }
VERSION : 0.1
// stored: AutoNumber true, IsIECCheckEnabled false, IsRetainMemResEnabled false, MemoryReserve 100, SetENOAutomatically false, UDAEnableTagReadback false
   VAR_OUTPUT
      blockDosing : Bool;
   END_VAR
   VAR RETAIN
      EnableMeasurment_TON { S7_SetPoint := 'True'} : TON_TIME;
      BlockDosing_TON { S7_SetPoint := 'True'} : TON_TIME;
   END_VAR
   VAR
      enableMeasureTime : Real;
      ChlorationCalculate { S7_SetPoint := 'True'} : "ChlorationCalculate";
      blockDosingTime : Real;
      R_TRIG { S7_SetPoint := 'True'} : R_TRIG;
   END_VAR
   VAR RETAIN
      Initial { S7_SetPoint := 'True'} : Bool := True;
   END_VAR
BEGIN
   IF "MB".Table.CycleDay >= "MB".Table.ChlorMeasureTable[3].CycleDay THEN
       #enableMeasureTime := "MB".Table.ChlorMeasureTable[3].MeasureTime;
       #blockDosingTime := "MB".Table.ChlorMeasureTable[3].BlockTime;
   ELSIF "MB".Table.CycleDay >= "MB".Table.ChlorMeasureTable[2].CycleDay THEN
       #enableMeasureTime := "MB".Table.ChlorMeasureTable[2].MeasureTime;
       #blockDosingTime := "MB".Table.ChlorMeasureTable[2].BlockTime;
   ELSIF "MB".Table.CycleDay >= "MB".Table.ChlorMeasureTable[1].CycleDay THEN
       #enableMeasureTime := "MB".Table.ChlorMeasureTable[1].MeasureTime;
       #blockDosingTime := "MB".Table.ChlorMeasureTable[1].BlockTime;
   ELSIF "MB".Table.CycleDay >= "MB".Table.ChlorMeasureTable[0].CycleDay THEN
       #enableMeasureTime := "MB".Table.ChlorMeasureTable[0].MeasureTime;
       #blockDosingTime := "MB".Table.ChlorMeasureTable[0].BlockTime;
   END_IF;

   #R_TRIG(CLK:="MB".Table.HMI_ChlorModeOn);

   IF #R_TRIG.Q THEN
       #ChlorationCalculate.doseCorection := 1;
       #ChlorationCalculate.doseCorectionOld := 1;
       #Initial := TRUE;
       "MB".Table.MeasureChanged := FALSE;
       RESET_TIMER(#EnableMeasurment_TON);
       RESET_TIMER(#BlockDosing_TON);
   END_IF;


   IF NOT "MB".Table.HMI_ChlorModeOn THEN
       "MB".Table.MeasureChanged := FALSE;
       RESET_TIMER(#EnableMeasurment_TON);
       RESET_TIMER(#BlockDosing_TON);
   END_IF;


   "MB".Table.TimeToMeasure := #enableMeasureTime - DINT_TO_REAL(#EnableMeasurment_TON.ET)/1000/60/60;
   "MB".Table.TimeToBlock := #blockDosingTime - DINT_TO_REAL(#BlockDosing_TON.ET)/1000/60/60;

   #blockDosing := #BlockDosing_TON.Q;
   "MB".Table.MeasureNotEntered := #blockDosing;

   "MB".Table.CriticalMeasureON := FALSE;

   IF "MB".Table.MeasuredChlor >= "MB".Table.CriticalMeasure THEN
       "MB".Table.CriticalMeasureON := TRUE;
       "MB".Table.ChlorationParams.ActualDose := 0;
   END_IF;

   IF "MB".Table.ChangeChlorMeasure THEN
       IF #EnableMeasurment_TON.Q OR #Initial THEN
           "MB".Table.MeasuredChlor := "MB".Table.ChlorMeasuredValue;
           #ChlorationCalculate(ChlorationParams := "MB".Table.ChlorationParams,
                                measuredChlorine := "MB".Table.ChlorMeasuredValue);
           "MB".Table.MeasureChanged := TRUE;
           RESET_TIMER(#EnableMeasurment_TON);
           RESET_TIMER(#BlockDosing_TON);
       END_IF;
       "MB".Table.ChangeChlorMeasure := FALSE;
       #Initial := FALSE;
       #BlockDosing_TON(IN := TRUE,
                        PT := REAL_TO_DINT(#blockDosingTime) * 1000 * 60*60);
       #EnableMeasurment_TON(IN := TRUE,
                             PT := REAL_TO_DINT(#enableMeasureTime) * 1000 * 60*60);
   END_IF;

   IF #EnableMeasurment_TON.Q THEN
       "MB".Table.MeasureChanged := FALSE;
   END_IF;
END_FUNCTION_BLOCK

FUNCTION_BLOCK "ChlorationCalculate"   // FB7, SCL
{ S7_Optimized_Access := 'TRUE' }
VERSION : 0.1
// stored: AutoNumber true, IsIECCheckEnabled false, IsRetainMemResEnabled false, MemoryReserve 100, SetENOAutomatically false, UDAEnableTagReadback false
   VAR_INPUT
      measuredChlorine : Real;
   END_VAR
   VAR_IN_OUT
      ChlorationParams : Struct
         SetpointMin : Real;
         SetpointMax : Real;
         BaseDose : Real;
         ActualDose : Real;
         DoseChangeMax : Real;
         DosingMin : Real;
         DosingMax : Real;
         CorectionCoef : Real;
      END_STRUCT;
   END_VAR
   VAR RETAIN
      setpointDeviation : Real;
      doseCorection : Real := 1.0;
      doseCorectionOld : Real := 1.0;
   END_VAR
   VAR
      doseChangeMaxReal : Real;
   END_VAR
BEGIN
   IF NOT "MB".Table.ChangeChlorMeasure THEN
       RETURN;
   END_IF;

   IF #measuredChlorine <= "MB".Table.Chlor_SetpointMin OR
       #measuredChlorine >= "MB".Table.Chlor_SetpointMax THEN

       #setpointDeviation := ((("MB".Table.Chlor_SetpointMax + "MB".Table.Chlor_SetpointMin) / 2) - #measuredChlorine)* "MB".Table.Chlor_Corection;

       #doseCorection := #doseCorectionOld * (1 + #setpointDeviation);

       #doseChangeMaxReal := #ChlorationParams.DoseChangeMax / 100;

       IF #doseCorection - #doseCorectionOld > #doseChangeMaxReal THEN
           #doseCorection := #doseCorectionOld * (1 + #doseChangeMaxReal);
       ELSIF #doseCorection - #doseCorectionOld < - (#doseChangeMaxReal) THEN
           #doseCorection := #doseCorectionOld * (1 - #doseChangeMaxReal);
       END_IF;

       #ChlorationParams.ActualDose := "MB".Table.Chlor_BaseDose * #doseCorection;

       IF #ChlorationParams.ActualDose >= #ChlorationParams.DosingMax THEN
           #doseCorection := #ChlorationParams.DosingMax / "MB".Table.Chlor_BaseDose;
           #ChlorationParams.ActualDose := "MB".Table.Chlor_BaseDose * #doseCorection;
       ELSIF #ChlorationParams.ActualDose <= #ChlorationParams.DosingMin THEN
           #doseCorection := #ChlorationParams.DosingMin / "MB".Table.Chlor_BaseDose;
           #ChlorationParams.ActualDose := "MB".Table.Chlor_BaseDose * #doseCorection;
       END_IF;

       #doseCorectionOld := #doseCorection;

   END_IF;
END_FUNCTION_BLOCK

ORGANIZATION_BLOCK "DayOn"   // OB10, SCL, TimeOfDay
{ S7_Optimized_Access := 'TRUE' }
VERSION : 0.1
// stored: AutoNumber true, IsIECCheckEnabled false, SetENOAutomatically false
   VAR_INPUT
      CaughtUp : Bool;   // OB call is caught up because time was set forward
      SecondTime : Bool;   // OB call is started a second time because time was set backward
   END_VAR
BEGIN
   IF "MB".Table.HMI_CycleOn THEN
       "MB".Table.CycleDay := "MB".Table.CycleDay + 1;
       IF "MB".Table.CycleDay = "MB".Table.CycleStartDay[0] THEN
           "MB".Table.UsePID := TRUE;
       END_IF;
       IF "MB".Table.CycleDay = "MB".Table.CycleStartDay[4] THEN
           "MB".Table.UsePID := FALSE;
       END_IF;

       IF "MB".Table.CycleDay = "MB".Table.ChlorationCounter_SwitchDay AND "MB".Table.ChlorationCounter_SwitchOn THEN
           "MB".Table.Chloration_ChooseCounter := 1;
       END_IF;
   END_IF;
   "MB".Table.DayChangeFlag := TRUE;
   "MB".Table.WaterCounterIn_DailyCount := 0;
   "MB".Table.WaterCounterOut_DailyCount := 0;
   "MB".Table.Doser1_DailyPulses := 0;
   "MB".Table.Doser2_DailyPulses := 0;
END_ORGANIZATION_BLOCK

ORGANIZATION_BLOCK "DiagnosticErrorInterrupt"   // OB82, LAD, DiagnosticErrorInterrupt
{ S7_Optimized_Access := 'TRUE' }
VERSION : 0.1
// stored: IsIECCheckEnabled false, SetENOAutomatically false
   VAR_INPUT
      IO_State : Word;   // IO state of the HW object
      LADDR : HW_ANY;   // Hardware identifier
      Channel : UInt;   // Channel number
      MultiError : Bool;   // =true if more than one error is present
   END_VAR
BEGIN
END_ORGANIZATION_BLOCK

ORGANIZATION_BLOCK "PullOrPlugOfModules"   // OB83, LAD, PullOrPlugOfModules
{ S7_Optimized_Access := 'TRUE' }
VERSION : 0.1
// stored: IsIECCheckEnabled false, SetENOAutomatically false
   VAR_INPUT
      LADDR : HW_IO;   // Hardware identifier
      Event_Class : Byte;   // 16#38/39: module inserted, removed
      Fault_ID : Byte;   // Fault identifier
   END_VAR
BEGIN
END_ORGANIZATION_BLOCK

ORGANIZATION_BLOCK "RackOrStationFailure"   // OB86, LAD, RackOrStationFailure
{ S7_Optimized_Access := 'TRUE' }
VERSION : 0.1
// stored: IsIECCheckEnabled false, SetENOAutomatically false
   VAR_INPUT
      LADDR : HW_DEVICE;   // Hardware identifier
      Event_Class : Byte;   // Event class
      Fault_ID : Byte;   // Fault identifier
   END_VAR
BEGIN
END_ORGANIZATION_BLOCK

FUNCTION "SystemClock" : Void   // FC1, SCL
{ S7_Optimized_Access := 'TRUE' }
VERSION : 0.1
// stored: AutoNumber true, IsIECCheckEnabled false, SetENOAutomatically false, UDAEnableTagReadback false
   VAR_TEMP
      Value : Int;
   END_VAR
BEGIN
   #Value := RD_SYS_T("Config".DateTime);
END_FUNCTION

FUNCTION_BLOCK "StepGenerator"   // FB22, SCL
{ S7_Optimized_Access := 'TRUE' }
VERSION : 0.1
// stored: AutoNumber true, IsIECCheckEnabled false, IsRetainMemResEnabled false, MemoryReserve 100, SetENOAutomatically false, UDAEnableTagReadback false
   VAR_INPUT
      Enable : Bool;
      Tanklevel : Real;
      TankLevelSetpoint : Real;
      KP : Real := 2.0;
      KI : Real := 0.2;
      KD : Real := 0.5;
      TI : Time := T#1s;
      LimitMin : Real := -100.0;
      LimitMax : Real := 100.0;
      DeadZone : Real := 1.0;
   END_VAR
   VAR_OUTPUT
      DamperPosition : Real;
   END_VAR
   VAR
      "e" : Real;
      PValue : Real;
      IValue : Real;
      DValue : Real;
      init : Bool;
      TopLevelSetPoint : Real;
      BottomlevelSetPoint : Real;
      PrevValue : Real;
      TON1 { S7_SetPoint := 'True'} : TON_TIME;
   END_VAR
BEGIN
   IF NOT #Enable THEN
       #init := false;
       #IValue := 0;
       #DValue := 0;
   END_IF;

   #TopLevelSetPoint := #TankLevelSetpoint + #DeadZone;
   #BottomlevelSetPoint := #TankLevelSetpoint - #DeadZone;

   #TON1(IN:=TRUE,
         PT:=#TI);



   IF #TON1.Q THEN
       IF #Tanklevel > #TopLevelSetPoint THEN
           #e := #e - #KP;
       ELSIF #Tanklevel < #BottomlevelSetPoint THEN
           #e := #e + #KP;
       END_IF;
       #DamperPosition := #e;
       RESET_TIMER(#TON1);
   END_IF;
END_FUNCTION_BLOCK

DATA_BLOCK "AIHandler_DB"   // DB4
VERSION : 0.1
// stored: AutoNumber true, DBAccessibleFromOPCUA true, InstanceOfName AIHandler, InstanceOfType FB
"AIHandler"
BEGIN
   TON1.PT := T#0MS;
   TON1.IN := FALSE;
   DelayTON.PT := T#0MS;
   DelayTON.IN := FALSE;
   FilterArray[0..199] := 0.0;
END_DATA_BLOCK

DATA_BLOCK "Alarms_DB"   // DB11
VERSION : 0.1
// stored: AutoNumber true, DBAccessibleFromOPCUA true, InstanceOfName Alarms, InstanceOfType FB
"Alarms"
BEGIN
   WaterOutMaxTON.PT := T#0MS;
   WaterOutMaxTON.IN := TRUE;
   WaterOutMinTON.PT := T#0MS;
   WaterOutMinTON.IN := TRUE;
END_DATA_BLOCK

DATA_BLOCK "ChlorMode_DB"   // DB6
VERSION : 0.1
// stored: AutoNumber true, DBAccessibleFromOPCUA true, InstanceOfName ChlorMode, InstanceOfType FB
"ChlorMode"
BEGIN
END_DATA_BLOCK

